	10:	//*****ClearUp****
		//Interpreter stoppen
		fbItpStartStopEx(bStart:= FALSE, bStop:= TRUE, sNciToPlc:= stGCodeRef.sNciToPlc);
		IF NOT fbItpStartStopEx.bBusy THEN
			IF fbItpStartStopEx.bErr THEN
				stError.ErrorId := UDINT_TO_UINT(fbItpStartStopEx.nErrId);
				nStateA_Common := 99;
			ELSE
				nStateA_Common := 11;
				fbFastMFunc.M_StopPrintAction(stGCodeRef.pCurrentTool,0);
				IF stGCodeRef.pCurrentTool > 0 THEN
					IF stGCodeRef.pCurrentTool^.P_eObjectType = E_ObjectType.OBJECTTYPE_VermesDisp THEN
						//Druck ausschalten
						MEMSET(ADR(stActionData),0,SIZEOF(stActionData));
						stActionData.eAction := E_Action.ACTION_SwitchPressure;
						stActionData.aParams[1] := 1;
						stGCodeRef.pCurrentTool^.M_ExeAction(stActionData);
					END_IF				
				END_IF
			END_IF
			IF pHighVoltTray > 0 THEN
				IF pHighVoltTray^.P_bPwrCutOffTriggered THEN
					nStateA_CommonNext := 30;	//In Parking-Pos fahren
				END_IF
				//Strom-Überwachung ausschalten
				pHighVoltTray^.M_CurrentMonitoring(FALSE);
			END_IF	
			fbItpStartStopEx(bStart:= FALSE, bStop:= FALSE, sNciToPlc:= stGCodeRef.sNciToPlc);
		END_IF
		
	11:	//Interpreter resetten (nötig, um Interpolationsgruppe zu löschen)
		fbItpResetEx2(bExecute:= TRUE, sNciToPlc:= stGCodeRef.sNciToPlc);
		IF NOT fbItpResetEx2.bBusy THEN
			IF fbItpResetEx2.bErr THEN
				stError.ErrorId := UDINT_TO_UINT(fbItpResetEx2.nErrId);
				nStateA_Common := 99;
			ELSE
				nStateA_Common := 20;
			END_IF
			fbItpResetEx2(bExecute:= FALSE, sNciToPlc:= stGCodeRef.sNciToPlc);
		END_IF
			
	20:	//Interpolationsgruppe löschen
		fbClearGroup(stGCodeRef:= stGCodeRef, bReGearInSlave:= TRUE, bExecute:= TRUE);
		IF NOT fbClearGroup.bBusy THEN
			IF fbClearGroup.bError THEN
				stError.ErrorId := fbClearGroup.nErrorId;
				nStateA_Common := 99;
			ELSE
				nStateA_Common := nStateA_CommonNext;
			END_IF
			fbClearGroup(stGCodeRef:= stGCodeRef, bExecute:= FALSE);
		END_IF
		
	30:	//In Parking-Pos fahren (MoveAllHome)
		MEMSET(ADR(stActionData),0,SIZEOF(stActionData));
		stActionData.eAction := E_Action.ACTION_MoveAllHome;
		stError.ErrorId := fbComplexAction.M_ExeAction(stActionData);
		IF stError.ErrorId > 0 THEN
			nStateA_Common := 99;
		ELSE
			nStateA_Common := 31;
		END_IF
		
	31: //MoveAllHome ready?
		IF NOT fbComplexAction.bBusy THEN
			IF fbComplexAction.bError THEN
				nStateA_Common := 99;
			ELSE
				nStateA_Common := 80;
			END_IF
		END_IF

END_CASE

IF nStateA_Common = 99 THEN
	stError.POUAction := E_POUACT.POUACT_A_Run;
	fbErrorList.M_Add(stError);
END_IF
END_ACTION

ACTION A_Start:
stError.POUState := nStateA_Common;

CASE nStateA_Common OF
	0:	//Interpolationsgruppe bilden
		stError.ErrorId := 0;
		fbBuildGroup(stGCodeRef:= stGCodeRef, bExecute:= TRUE);
		IF NOT fbBuildGroup.bBusy THEN
			IF fbBuildGroup.bError THEN
				stError.ErrorId := fbBuildGroup.nErrorId;
				nStateA_Common := 99;
			ELSE
				nStateA_Common := 1;
			END_IF
			fbBuildGroup(stGCodeRef:= stGCodeRef, bExecute:= FALSE);
		END_IF
		
		//Tools iterieren, in ToolAssigTable eintragen und gleich das MES-Tool ermitteln, welches im nächsten Schritt
		//eventuell vom Freifahren ausgeschlossen wird
	1:  pGCodeTool := 0;
		pMesCartDisp := 0;
		pHighVoltTray := pTarget^.M_GetFirstParentOfType(E_ObjectType.OBJECTTYPE_HighVoltTray);
		memset(ADR(GCode.stGCodeRef.aToolTable),0, SIZEOF(ST_GCodeTool) * GCode.cMaxGCodeTools);
		stGCodeRef.pHead^.P_pObjCollectNode^.nodes.M_GetIterator(iterDeep);
		WHILE iterDeep.pNode > 0 DO
			IF iterDeep.pNode^.P_pObject > 0 AND_THEN iterDeep.pNode^.P_pObject^.M_bIsGroup(E_ObjectGroup.OBJECTGROUP_MzTool) THEN
				pTempTool := iterDeep.pNode^.P_pObject;
				IF fbObjectDirectory.M_ObjIsGCodeTool(pTempTool^.P_nObjectID) THEN //GCodeTool?
					pGCodeTool := pTempTool;
					IF pGCodeTool^.P_nGCodeToolNr > 0 THEN
						IF pGCodeTool^.P_nGCodeToolNr <= cMaxGCodeTools THEN
							IF stGCodeRef.aToolTable[pGCodeTool^.P_nGCodeToolNr].pMzTool = 0 THEN
								stGCodeRef.aToolTable[pGCodeTool^.P_nGCodeToolNr].pMzTool := pGCodeTool;
								//MES-Kartusche und MES-Tray vorhanden?
								IF (pGCodeTool^.P_eObjectType = E_ObjectType.OBJECTTYPE_CartDispenser OR
									pGCodeTool^.P_eObjectType = E_ObjectType.OBJECTTYPE_CartDispStirrer) AND pHighVoltTray > 0 THEN
									pMesCartDisp := pGCodeTool;
									IF NOT pMesCartDisp^.P_bIsMESTool THEN
										//befindet sich MES-Kartusche über MES-Tray? Diese würde vom Freifahren ausgeschlossen
										IF NOT F_PointInnerRect(pMesCartDisp^.P_stCurrentPosPhys,pHighVoltTray^.P_stAbsRect) THEN
											pMesCartDisp := 0;	
										END_IF
									END_IF
								END_IF
								//Checken, ob Tool bereit für den Start im GCode-Mode
								stError.ErrorId := pGCodeTool^.M_CheckGCodeStart();
								IF stError.ErrorId > 0 THEN
									stError.ObjectId := pGCodeTool^.P_nObjectID;
									EXIT;
								END_IF
							ELSE
								//schon belegt, zwei Tools haben die gleiche ToolNr
								//sollte eigentlich schon in der GUI abgefangen werden
								stError.ErrorId := E_ErrorIdGCode.ERRORID_InvalidToolNr;
								EXIT;			
							END_IF
						ELSE
							//ToolNr zu groß
							//sollte eigentlich schon in der GUI abgefangen werden
							stError.ErrorId := E_ErrorIdGCode.ERRORID_InvalidToolNr;
							EXIT;			
						END_IF
					END_IF					
				END_IF
			END_IF
			iterDeep.M_Increment();
		END_WHILE
		
		//GCodeTargetNummern in TargetTable eintragen
		memset(ADR(GCode.stGCodeRef.aTargetTable),0, SIZEOF(UINT) * GCode.cMaxGCodeTargets);
		//wie komme ich hier an die Workplate ran?
		//über den Head und die zugeordnete Workplate
		stGCodeRef.pHead^.P_pAssignWorkplate^.P_pObjCollectNode^.nodes.M_GetIterator(iterDeep);
		WHILE iterDeep.pNode > 0 DO
			(* 1. Finde ein Objekt im Tree 2. Muss ein mögliches Target sein 3. Diese Objekt muss die gleiche Obj Id haben wie der in der GUI ausgewählte Print Point *)
			IF iterDeep.pNode^.P_pObject > 0  AND_THEN iterDeep.pNode^.P_pObject^.M_bIsGroup(E_ObjectGroup.OBJECTGROUP_Target) AND iterDeep.pNode^.P_pObject^.P_nObjectID = stInfo2.nTargetObjId THEN
				pTarget := iterDeep.pNode^.P_pObject;
				IF pTarget^.P_nGCodeTargetNr > 0 THEN
					//darf nicht größe als 20 sein 
					IF  pTarget^.P_nGCodeTargetNr > GCode.cMaxGCodeTargets THEN
						{warnig 'Imlement proper ErrorID'}
						stError.ErrorId := E_ErrorIdGCode.ERRORID_InvalidToolNr;
						RETURN;
					END_IF
					//darf noch nicht belegt sein
					IF GCode.stGCodeRef.aTargetTable[pTarget^.P_nGCodeTargetNr] > 0 THEN
						{warnig 'Imlement proper ErrorID'}
						stError.ErrorId := E_ErrorIdGCode.ERRORID_InvalidToolNr;
						RETURN;
					END_IF
					GCode.stGCodeRef.aTargetTable[pTarget^.P_nGCodeTargetNr] := pTarget^.P_nObjectID;
				END_IF
			END_IF
			iterDeep.M_Increment();
		END_WHILE
	
		//Tools freifahren
		IF stError.ErrorId = 0 THEN
			stError.ErrorId := stGCodeRef.pHead^.M_MoveFree(pMesCartDisp);
			IF stError.ErrorId > 0 THEN
				stError.ObjectId := stGCodeRef.pHead^.P_nObjectID;
				nStateA_Common := 99;
			ELSE
				nStateA_Common := 2;
			END_IF
		ELSE
			nStateA_Common := 99;
		END_IF
	
	2:	//Tools frei?
		IF NOT stGCodeRef.pHead^.M_GetActionBusy(E_Action.ACTION_MoveZ) THEN
			nStateA_Common := 3;
		END_IF
		
		IF stGCodeRef.pHead^.P_bError THEN
			stError.ErrorId := stGCodeRef.pHead^.P_nErrorId;
			stError.ObjectId := stGCodeRef.pHead^.P_nObjectID;
			nStateA_Common := 99;
		END_IF
	
	3:	//XY-Nullpunktverschiebung schreiben
		fbItpWriteZeroShiftEx(bExecute:= TRUE, sNciToPlc:= stGCodeRef.sNciToPlc, nZsNo:= 54, sZeroShiftDesc:= stGCodeRef.sZeroShiftDesc);	
		IF NOT fbItpWriteZeroShiftEx.bBusy THEN
			IF fbItpWriteZeroShiftEx.bErr THEN
				stError.ErrorId := UDINT_TO_UINT(fbItpWriteZeroShiftEx.nErrId);
				nStateA_Common := 99;
			ELSE
				stGCodeRef.pCurrentTool := 0;
				fbFastMFunc.M_Reset();
				fbHskMFunc.M_Reset();
				nStateA_Common := 4;
			END_IF
			fbItpWriteZeroShiftEx(bExecute:= FALSE, sNciToPlc:= GCode.stGCodeRef.sNciToPlc, nZsNo:= 54, sZeroShiftDesc:= stGCodeRef.sZeroShiftDesc);
		END_IF
		
	4: //RParameter 101 bis 125 löschen
		fbItpWriteRParams(bExecute:= TRUE, pAddr:= ADR(aRParamInit), nIndex:= 101 , nCount:= 25, sNciToPlc:= stGCodeRef.sNciToPlc); 
		IF NOT fbItpWriteRParams.bBusy THEN
			fbItpWriteRParams(bExecute:= FALSE, sNciToPlc:= stGCodeRef.sNciToPlc);
			lrAngle := pTarget^.P_lrAbsAngle;
			stGCodeRef.fbLimitCuboid.P_lrAngle := lrAngle;
			nStateA_Common := 5;
		END_IF
		
	5: //Verdrehwinkel des Targets in R126 schreiben (Winkel wird einen Schritt vorher ermittelt
		fbItpWriteRParams(bExecute:= TRUE, pAddr:= ADR(lrAngle), nIndex:= 126 , nCount:= 1, sNciToPlc:= stGCodeRef.sNciToPlc);
		IF NOT fbItpWriteRParams.bBusy THEN
			fbItpWriteRParams(bExecute:= FALSE, sNciToPlc:= stGCodeRef.sNciToPlc);
			nStateA_Common := 6;
		END_IF

	6:	//Interpreter starten
		fbItpStartStopEx(bStart:= TRUE,	bStop:= FALSE, sNciToPlc:= GCode.stGCodeRef.sNciToPlc);
		IF NOT fbItpStartStopEx.bBusy THEN
			IF fbItpStartStopEx.bErr THEN
				stError.ErrorId := UDINT_TO_UINT(fbItpStartStopEx.nErrId);
				nStateA_Common := 99;
			ELSE
				nStateA_Common := 7;
			END_IF
			fbItpStartStopEx(bStart:= FALSE, bStop:= FALSE, sNciToPlc:= GCode.stGCodeRef.sNciToPlc);
		END_IF
END_CASE

IF nStateA_Common = 7 THEN
	//Abfrage  des InterpreterStatus
	//Wechsel des States von Ready auf einen anderen State -> weiter zu A_Running
	//Nach dem Laden des Programms geht der Interpreter in Ready
	stInfo.nNciState := ItpGetStateInterpreter(GCode.stGCodeRef.sNciToPlc);
	IF stInfo.nNciState <> Tc2_NCI.NCI_INTERPRETER_READY THEN
		IF pHighVoltTray > 0 THEN
			//Strom-Überwachung einschalten
			pHighVoltTray^.M_CurrentMonitoring(TRUE);
		END_IF
		stGCodeRef.lrNcOverride := 100.0;
		nStateA_Common := 80;
	END_IF
END_IF

//Achtung, Implementation von Cancel ist hier schon wichtig!!!

IF nStateA_Common = 99 THEN
	stError.POUAction := E_POUACT.POUACT_A_Start;
	fbErrorList.M_Add(stError);
END_IF
END_ACTION

METHOD M_ClearGroup : ST_MethResult

VAR_INPUT
	bReGearIn : BOOL;
END_VAR
IF pXDrive = 0 OR pYDrive = 0 THEN	//GCode-Modul wurde noch nicht gestartet und folglich kann auch keine Gruppe vorhanden sein
	RETURN;
END_IF
M_ClearGroup.bBusy := TRUE;
fbClearGroup(stGCodeRef:= stGCodeRef, bReGearInSlave:= bReGearIn, bExecute:= TRUE);
IF NOT fbClearGroup.bBusy THEN
	IF fbClearGroup.bError THEN
		M_ClearGroup.bError := TRUE;
		M_ClearGroup.nErrorId := fbClearGroup.nErrorId;
	END_IF
	M_ClearGroup.bBusy := FALSE;
	fbClearGroup(stGCodeRef:= stGCodeRef, bExecute:= FALSE);
END_IF
END_METHOD

METHOD M_Continue : ERRORID
VAR_INPUT
END_VAR
IF nState = 6 THEN
	eGCodeState := E_GCodeState.GCodeState_ContinueRequest;
	nState := 7;
END_IF
END_METHOD

METHOD M_Pause : ERRORID
VAR_INPUT
END_VAR
IF stInfo.eGCodeState = E_GCodeState.GCodeState_Running AND nStateA_Common = 0 THEN
	IF pHighVoltTray > 0 THEN
		//Strom-Überwachung ausschalten
		pHighVoltTray^.M_CurrentMonitoring(FALSE);
	END_IF
	nState := 5;
END_IF
END_METHOD

METHOD M_Reset
VAR_INPUT
END_VAR
IF nState = 99 THEN
	nState := 60;
END_IF
END_METHOD

METHOD M_SetSequenceIds
VAR_INPUT
	pIdArray : POINTER TO ARRAY[1..5] OF DINT;
END_VAR
MEMCPY(ADR(stGCodeRef.aSequenceIds),pIdArray,20);
END_METHOD

METHOD M_SetStartZeroPoint : ERRORID
VAR_INPUT
	nTargetObjId 	: UINT;
	eTargetRef		: E_TargetRef;
	nCol			: UINT;
	nRow			: UINT;
	nZOffset		: DINT;
	nPausePointObjId: UINT;
	rHeight			: REAL;
END_VAR

VAR
	pMtp		: POINTER TO FB_Mtp;
	stPosTemp	: ST_3DPoint;
	rHeightTemp	: REAL;
END_VAR
CASE fbObjectDirectory.M_GetObjType(nTargetObjId) OF
	E_ObjectType.OBJECTTYPE_Point, E_ObjectType.OBJECTTYPE_Slide:
		//als TargetRef wird hier immer Mitte angenommen
		pTarget := fbObjectDirectory.M_GetObjPointer(nTargetObjId);
		stGCodeRef.stStartPos := pTarget^.M_GetAbsPos(0,E_TargetRef.TARGETREF_Center,0,0,0,1,nErrorId=> M_SetStartZeroPoint);
		GCode.stInfo2.nTargetObjId := nTargetObjId;
		
	E_ObjectType.OBJECTTYPE_Mtp:
		pTarget := fbObjectDirectory.M_GetObjPointer(nTargetObjId);
		IF eTargetRef <> E_TargetRef.TARGETREF_TwoDimArray THEN
			M_SetStartZeroPoint := E_ErrorIdCmd.ERRORID_InvalidTargetPointRef;
			RETURN;
		END_IF
		pMtp := pTarget;
		stGCodeRef.stStartPos := pMtp^.M_GetAbsPos(0,eTargetRef, nCol, nRow, 0, 1, nErrorId=> M_SetStartZeroPoint);
		IF M_SetStartZeroPoint > 0 THEN
			RETURN;
		END_IF
ELSE
	M_SetStartZeroPoint := E_ErrorIdCmd.ERRORID_UnsuitableTarget;
	RETURN;
END_CASE

stGCodeRef.fbLimitCuboid.P_stRefPoint := stGCodeRef.stStartPos;

stGCodeRef.pWaitPoint := 0;
IF nPausePointObjId > 0 THEN
	IF fbObjectDirectory.M_GetObjType(nPausePointObjId) = E_ObjectType.OBJECTTYPE_Point THEN
		stGCodeRef.pWaitPoint := fbObjectDirectory.M_GetObjPointer(nPausePointObjId);
	ELSE
		M_SetStartZeroPoint := E_ErrorIdGCode.ERRORID_InvalidPausePoint;
		RETURN;
	END_IF
END_IF

//Es kann nur der obere Head GCode ausführen
stGCodeRef.pHead := fbObjectDirectory.M_GetTopHead();

pXDrive := stGCodeRef.pHead^.P_pXDrive;
pYDrive := stGCodeRef.pHead^.P_pYDrive;

//Da hier noch kein Tool ausgewählt ist, bezieht sich Nullpunktverschiebung in XY bezieht sich vorerst den Head
//Bei der Toolauswahl wird entsprechend verrechnet 
stPosTemp := F_Sub3DPoints(stGCodeRef.stStartPos, stGCodeRef.pHead^.P_stAbsPosTotal);
stGCodeRef.sZeroShiftDesc.fShiftX := stPosTemp.X / 1000.0;
stGCodeRef.sZeroShiftDesc.fShiftY := stPosTemp.Y / 1000.0;
stGCodeRef.sZeroShiftDesc.fShiftZ := (stGCodeRef.stStartPos.Z + DINT_TO_REAL(nZOffset)) / 1000.0;
END_METHOD

METHOD M_ShiftZPos : ERRORID
VAR_INPUT
	rValue : REAL;
END_VAR
//Wird nur verschoben, wenn in Running oder Pause
IF (NOT bWriteZeroShift) AND (eGCodeState = E_GCodeState.GCodeState_Running OR eGCodeState = E_GCodeState.GCodeState_Pause) THEN
	stGCodeRef.sZeroShiftDesc.fShiftZ := stGCodeRef.sZeroShiftDesc.fShiftZ + (rValue / 1000.0);
	bWriteZeroShift := TRUE;
END_IF
END_METHOD

METHOD M_Start : ERRORID
VAR_INPUT
	sFileNumber : STRING;
END_VAR
//Kann nur aus dem State "Idle" ausgeführt werden
IF stInfo.eGCodeState = E_GCodeState.GCodeState_Idle THEN
	{IF defined(WIN10)}
	sGCodeFile := CONCAT(cPathWIN_10, sFileNumber);
	{ELSE}
	sGCodeFile := CONCAT(cPathWIN_EMBEDDED, sFileNumber);
	{END_IF}
	sGCodeFile := CONCAT(sGCodeFile,'.nc');
	bStop := FALSE;
	nState := 2;
	stInfo.eGCodeState := eGCodeState := E_GCodeState.GCodeState_Loading;
	stInfo.nFileNr := STRING_TO_UDINT(sFileNumber);
ELSE
	M_Start := E_ErrorIdGCode.ERRORID_InvalidNciState;
END_IF
END_METHOD

METHOD M_Stop
VAR_INPUT
END_VAR
IF nState > 1 THEN //Idle
	bStop := TRUE;
END_IF
END_METHOD

PROPERTY P_bMoveActionsLocked : BOOL
GET
P_bMoveActionsLocked := bMoveActionsLocked;
END_GET
SET
bMoveActionsLocked := P_bMoveActionsLocked;
END_SET
END_PROPERTY

PROPERTY P_bNciAvailable : BOOL
GET
P_bNciAvailable := bNciAvailable;
END_GET
END_PROPERTY

PROPERTY P_nProgress : UINT
GET
P_nProgress := nProgress;
END_GET
END_PROPERTY

END_PROGRAM

// ---- Hardware/XYDrive/FB_XYDriveBase.TcPOU
FUNCTION_BLOCK FB_XYDriveBase EXTENDS FB_HwModule
VAR PERSISTENT
	rRefPosMaster		: REAL;
	rWorkplateLength 	: REAL;
	rNullPosDist 		: REAL;
	rMaxPosDist 		: REAL;
	rSetupPosDist 		: REAL;
	rLimitMargeNeg 		: REAL;
	rLimitMargePos 		: REAL;
	rMaxSpeed 			: REAL;
	bSetupOK 			: BOOL; //Setup wurde durchgeführt	
	bInvertInitDir 		: BOOL; //Richtung bei Initialisierung umkehren(negativ)
END_VAR

VAR
	nErrorId 			: ERRORID;
	rActPos				: REAL;
	bHomed				: BOOL;
	
	eXYOrientation		: E_XYOrientation;

	bWriteAxisParameter : BOOL;
	nStateA_WriteAxisParamter : USINT;
	nStateWriteLimitNegative : USINT;
	nStateWriteLimitPositive : USINT;
	nStateWriteNCIFastSpeed : USINT;

	bSetup : BOOL;
	nStateA_Setup : USINT;
	bSetupWaitForResp : BOOL;
	bContinueSetup : BOOL;
	bSetupError: BOOL;
	
	bInit : BOOL;
	nStateA_Init : USINT;
	bReInit : BOOL;
	rHomePos : REAL;
	Delay : TON;
	bStopInit : BOOL;
	
	bJog : BOOL;
	nStateA_Jog : USINT;
	bJogForward : BOOL;
	bJogBackward : BOOL;
	bJogInching : BOOL;
	tmrJog : TON;	
	
	bMoveAbs : BOOL;
	nStateMoveAbs : USINT;
	bMoveRel : BOOL;
	nStateMoveRel : USINT;
	
	bCapture : BOOL;
	nStateA_Capture : USINT;
	bStopCapture : BOOL;
	nStateA_StopCapture : USINT;
	bCaptureOk 			: BOOL;
	bCaptureStopped 	: BOOL;
	rCapturedPos		: REAL;
	
	bStop	: BOOL;
	nStateA_Stop : USINT;
	
	bReset : BOOL;
	nStateA_Reset : USINT;
	
	nStateA_Error : USINT;
	
	pMultiZRef : POINTER TO FB_MultiZRef;
	
	stAdsAddress : ST_AdsAdress;
	
	rTrigError	: R_TRIG;

END_VAR


IF bWriteAxisParameter THEN
	A_WriteAxisParameter();
	IF nStateA_WriteAxisParamter >= 80 THEN
		IF nStateA_WriteAxisParamter >= 99 THEN
			bError := TRUE;
		END_IF
		nStateA_WriteAxisParamter := 0;
		bWriteAxisParameter := FALSE;
	END_IF
END_IF

IF bSetup THEN
	A_Setup();
	IF nStateA_Setup >= 80 THEN
		IF nStateA_Setup >= 99 THEN
			bError := TRUE;
		END_IF
		nStateA_Setup := 0;
		bSetup := FALSE;
	END_IF
END_IF

IF bInit THEN
	A_Init();
	IF nStateA_Init = 80 THEN
		nStateA_Init := 0;
		bInit := FALSE;
	END_IF

	IF nStateA_Init = 99 THEN	//Error
		nStateA_Init := 0;
		bInit := FALSE;
		bError := TRUE;
	END_IF
END_IF

IF bMoveAbs THEN
	A_MoveAbs();
	IF nStateMoveAbs >= 80 THEN
		IF nStateMoveAbs >= 99 THEN	//Error
			bError := TRUE;
		END_IF
		nStateMoveAbs := 0;
		bMoveAbs := FALSE;
	END_IF	
END_IF

IF bMoveRel THEN
	A_MoveRel();
	IF nStateMoveRel >= 80 THEN
		IF nStateMoveRel >= 99 THEN	//Error
			bError := TRUE;
		END_IF
		nStateMoveRel := 0;
		bMoveRel := FALSE;
	END_IF	
END_IF

IF bJog THEN
	A_Jog();
	IF nStateA_Jog >= 80 THEN
		IF nStateA_Jog >= 99 THEN	//Error
			bError := TRUE;
		END_IF
		nStateA_Jog := 0;
		bJog := FALSE;
	END_IF	
END_IF

IF bCapture THEN
	A_Capture();
	IF nStateA_Capture >= 80 THEN
		IF nStateA_Capture >= 99 THEN	//Error
			bError := TRUE;
		END_IF
		nStateA_Capture := 0;
		bCapture := FALSE;
	END_IF	
END_IF

IF bStopCapture THEN
	A_StopCapture();
	IF nStateA_StopCapture >= 80 THEN
		IF nStateA_StopCapture >= 99 THEN	//Error
			bError := TRUE;
		END_IF
		nStateA_StopCapture := 0;
		bStopCapture := FALSE;
	END_IF	
END_IF

IF bReset THEN
	A_Reset();
	IF nStateA_Reset >= 80 THEN
		IF nStateA_Reset >= 99 THEN
			bError := TRUE;
		END_IF
		nStateA_Reset := 0;
		bReset := FALSE;
	END_IF
END_IF

IF bError THEN
	A_Error();
END_IF

IF NOT (bInit OR bMoveAbs OR bMoveRel OR bJog OR bReset OR bSetup) THEN
	bStop := FALSE;
	bBusy := FALSE;
ELSE
	bBusy := TRUE;
END_IF

rTrigError(CLK:= bError);
IF rTrigError.Q THEN
	stError.ErrorId := nErrorId;
	fbErrorList.M_Add(stError);
END_IF

PROPERTY P_bHomed : BOOL
GET
P_bHomed := bHomed;
END_GET
END_PROPERTY

ACTION A_Setup:

END_ACTION

METHOD M_GetProperty : ERRORID
VAR_INPUT
	eType	: E_HardwarePropType;
END_VAR
VAR_OUTPUT
	nValue 	: DINT;
END_VAR
CASE eType OF
	E_HardwarePropType.RefPos1:
		nValue := REAL_TO_DINT(rRefPosMaster);
	E_HardwarePropType.MinPos:
		nValue := REAL_TO_DINT(P_rMinPos);
	E_HardwarePropType.MaxPos:
		nValue := REAL_TO_DINT(P_rMaxPos);
	E_HardwarePropType.LimitMargeNeg:
		nValue := REAL_TO_DINT(rLimitMargeNeg);
	E_HardwarePropType.LimitMargePos:
		nValue := REAL_TO_DINT(rLimitMargePos);
	E_HardwarePropType.MaxSpeed:
		nValue := REAL_TO_DINT(rMaxSpeed);
	E_HardwarePropType.WorkplateDim:
		nValue := REAL_TO_DINT(rWorkplateLength);
	E_HardwarePropType.NullPosDist:
		nValue := REAL_TO_DINT(rNullPosDist);
	E_HardwarePropType.MaxPosDist:
		nValue := REAL_TO_DINT(rMaxPosDist);
	E_HardwarePropType.SetupPosDist:
		nValue := REAL_TO_DINT(rSetupPosDist);
	E_HardwarePropType.InvertInitDir:
		nValue := BOOL_TO_DINT(bInvertInitDir);		
ELSE
	M_GetProperty := E_ErrorIdCmd.ERRORID_InvalidHwProperty;	
END_CASE
END_METHOD

METHOD M_Init : ERRORID
VAR_INPUT
	bReInit : BOOL;
END_VAR
IF bBusy THEN
	M_Init := E_ErrorIdCmd.ERRORID_AxisStillBusy;
ELSE
	THIS^.bReInit := bReInit;
	//Die Action wird von hier aus einmalig ausgeführt damit ein Aufruf schon in diesem Zyklus stattfindet
	rHomePos := rRefPosMaster;
	bInit := TRUE;
	A_Init();		
END_IF
END_METHOD

METHOD M_PowerOn : ERRORID
VAR_INPUT
END_VAR
END_METHOD

METHOD M_MoveRel : ERRORID
VAR_INPUT
	rDistance		: REAL;
	rSpeed			: REAL;
	rAcceleration 	: REAL;
	rDeceleration 	: REAL;	
END_VAR
END_METHOD

ACTION A_Reset:

END_ACTION

PROPERTY P_bIsTwinDrive : BOOL
GET
END_GET
END_PROPERTY

METHOD M_Stop : ERRORID
VAR_INPUT
END_VAR
IF bBusy AND NOT bStop THEN
	bStop := TRUE;
END_IF
END_METHOD

METHOD M_Setup : ERRORID
VAR_INPUT
END_VAR
IF bBusy THEN
	M_Setup := E_ErrorIdCmd.ERRORID_AxisStillBusy;
ELSE
	THIS^.bReInit := TRUE;
	rHomePos := 0;
	bSetup := TRUE;
END_IF
END_METHOD

PROPERTY P_nErrorId : ERRORID
GET
P_nErrorId := nErrorId;
END_GET
END_PROPERTY

METHOD M_PowerOff : ERRORID
VAR_INPUT
END_VAR
END_METHOD

PROPERTY P_bIsMoving : BOOL
GET
END_GET
END_PROPERTY

ACTION A_Error:

END_ACTION

PROPERTY P_pAxisRef : POINTER TO AXIS_REF
GET
END_GET
END_PROPERTY

ACTION A_Init:

END_ACTION

METHOD M_StopCapture : ERRORID
VAR_INPUT
END_VAR
bStopCapture := TRUE;
bCaptureStopped := FALSE;
A_StopCapture();
END_METHOD

METHOD M_SetProperty : ERRORID
VAR_INPUT
	eType	: E_HardwarePropType;
	nValue 	: DINT;
END_VAR
CASE eType OF
	E_HardwarePropType.RefPos1:
		rRefPosMaster := DINT_TO_REAL(nValue);
	E_HardwarePropType.MinPos:
		M_SetProperty := E_ErrorIdCmd.ERRORID_OnlyReadHwProp;
	E_HardwarePropType.MaxPos:
		M_SetProperty := E_ErrorIdCmd.ERRORID_OnlyReadHwProp;
	E_HardwarePropType.LimitMargeNeg:
		rLimitMargeNeg := DINT_TO_REAL(nValue);
		bWriteAxisParameter := TRUE;
	E_HardwarePropType.LimitMargePos:
		rLimitMargePos := DINT_TO_REAL(nValue);
		bWriteAxisParameter := TRUE;
	E_HardwarePropType.MaxSpeed:
		rMaxSpeed := DINT_TO_REAL(nValue);
		bWriteAxisParameter := TRUE;
	E_HardwarePropType.WorkplateDim:
		rWorkplateLength := DINT_TO_REAL(nValue);
		bWriteAxisParameter := TRUE;
	E_HardwarePropType.NullPosDist:
		rNullPosDist := DINT_TO_REAL(nValue);
		bWriteAxisParameter := TRUE;
	E_HardwarePropType.MaxPosDist:
		rMaxPosDist := DINT_TO_REAL(nValue);
		bWriteAxisParameter := TRUE;
	E_HardwarePropType.SetupPosDist:
		rSetupPosDist := DINT_TO_REAL(nValue);
	E_HardwarePropType.InvertInitDir:
		bInvertInitDir := DINT_TO_BOOL(nValue);
ELSE
	M_SetProperty := E_ErrorIdCmd.ERRORID_InvalidHwProperty;	
END_CASE
END_METHOD

METHOD M_GearOut : ST_MethResult
END_METHOD

PROPERTY P_tHomingTime : TIME
GET
//nur aus Kompatibilitätsgründen PlattformD impl.
P_tHomingTime := T#0s;
END_GET
END_PROPERTY

METHOD M_Capture : ERRORID
VAR_INPUT
END_VAR
END_METHOD

PROPERTY P_stAdsAddress : ST_AdsAdress
SET
stAdsAddress := P_stAdsAddress;
END_SET
GET
P_stAdsAddress := stAdsAddress;
END_GET
END_PROPERTY

PROPERTY P_bHasJob : BOOL
GET
END_GET
END_PROPERTY

PROPERTY P_bCoupled : BOOL
GET
END_GET
END_PROPERTY

ACTION A_Capture:

END_ACTION

PROPERTY P_bHoming : BOOL
GET
P_bHoming := bInit;
END_GET
END_PROPERTY

PROPERTY P_bSetupWaitForResp : BOOL
GET
P_bSetupWaitForResp := bSetupWaitForResp;
END_GET
END_PROPERTY

METHOD FB_init : BOOL
VAR_INPUT
	bInitRetains 	: BOOL; // if TRUE, the retain variables are initialized (warm start / cold start)
	bInCopyCode 	: BOOL;  // if TRUE, the instance afterwards gets moved into the copy code (online change)
	eXYOrientation	: E_XYOrientation;
END_VAR
THIS^.eXYOrientation := eXYOrientation;
END_METHOD

METHOD M_Reset
VAR_INPUT
END_VAR
IF bError AND NOT bReset THEN
	bReset := TRUE;
END_IF
END_METHOD

ACTION A_StopCapture:

END_ACTION

METHOD M_ContinueSetup
VAR_INPUT
END_VAR
bContinueSetup := TRUE;
END_METHOD

ACTION A_WriteAxisParameter:

END_ACTION

PROPERTY P_rActPos : REAL
GET
P_rActPos := rActPos;
END_GET
END_PROPERTY

PROPERTY P_rMaxPos : REAL
GET
P_rMaxPos := rWorkplateLength - rNullPosDist - rMaxPosDist - rLimitMargePos;
END_GET
END_PROPERTY

METHOD M_Jog : ERRORID
VAR_INPUT
	bForward	: BOOL;
	bBackward	: BOOL;
	bInching	: BOOL;
	rDistance	: REAL;
	rSpeed		: REAL;		
END_VAR
END_METHOD

ACTION A_Jog:

END_ACTION

ACTION A_MoveRel:

END_ACTION

PROPERTY P_rMinPos : REAL
GET
P_rMinPos := rLimitMargeNeg;
END_GET
END_PROPERTY

METHOD M_MoveAbs : ERRORID
VAR_INPUT
	rPosition 		: REAL;
	rSpeed			: REAL;
	rAcceleration 	: REAL;
	rDeceleration 	: REAL;
END_VAR
END_METHOD

PROPERTY P_bCaptureOk : BOOL
GET
P_bCaptureOk := bCaptureOk;
END_GET
END_PROPERTY

METHOD M_GearIn : ST_MethResult
END_METHOD

PROPERTY P_pMultiZRef : POINTER TO FB_MultiZRef
SET
pMultiZRef := P_pMultiZRef;
END_SET
GET
P_pMultiZRef := pMultiZRef;
END_GET
END_PROPERTY

PROPERTY P_rMaxSpeed : REAL
GET
P_rMaxSpeed := rMaxSpeed;
END_GET
END_PROPERTY

METHOD M_SetProperties : ERRORID
VAR_INPUT
	refCmdData : REFERENCE TO ST_CmdData;
END_VAR
rWorkplateLength := DINT_TO_REAL(refCmdData.n32Data[1]);
rNullPosDist := DINT_TO_REAL(refCmdData.n32Data[2]);
rMaxPosDist := DINT_TO_REAL(refCmdData.n32Data[3]);
rSetupPosDist := DINT_TO_REAL(refCmdData.n32Data[4]);
bInvertInitDir := DINT_TO_BOOL(refCmdData.n32Data[5]);
END_METHOD

ACTION A_MoveAbs:

END_ACTION

PROPERTY P_rCapturedPos : REAL
GET
P_rCapturedPos := rCapturedPos;
END_GET
END_PROPERTY

PROPERTY P_bCaptureStopped : BOOL
GET
P_bCaptureStopped := bCaptureStopped;
END_GET
END_PROPERTY

PROPERTY P_bIsCoupled : BOOL
GET
END_GET
END_PROPERTY

PROPERTY P_eXYOrientation : E_XYOrientation
GET
P_eXYOrientation := eXYOrientation;
END_GET
SET
eXYOrientation := P_eXYOrientation;
END_SET
END_PROPERTY

END_FUNCTION_BLOCK

// ---- Hardware/MultiZ/FB_MultiZRef.TcPOU
FUNCTION_BLOCK FB_MultiZRef EXTENDS FB_CanNodeBase

VAR_INPUT
	aFbZAxisRef 	: ARRAY[1..7] OF FB_ZAxisRef(THIS);
	aFbPiezoRef		: ARRAY[1..7] OF FB_PiezoRef(THIS);
	aFbHeaterRef	: ARRAY[1..7] OF FB_MZHeaterRef(THIS);
	aFbExtruderRef	: ARRAY[1..7] OF FB_PistonExtruderRef(THIS);
	aFbGripperRef	: ARRAY[1..7] OF FB_GripperRef(THIS);
	stStampSupport 	: ST_StampSupport;
	stStrobTrigger	: ST_StrobTrigger; //Sdo
	aDigiOut		AT %Q* : ARRAY[1..7] OF BOOL;
	aFbGPInputRef	: ARRAY[1..6] OF FB_GPInputRef(THIS);
	bFixConfig		: BOOL;
	nErrorGlobal	AT %I* : USINT;
END_VAR

VAR
	i				: USINT;
	bLegacy			: BOOL;
	nAxisNr			: USINT;
	nAxisNrZSensor 	: USINT;
	
	//bPrepareAxis 			: BOOL;
	nStateA_PrepareAxis 	: USINT;
	nStateA_PrepareAxisNext : USINT;
	nPrepareAxisNr 			: USINT;
	nTemp					: UDINT;
	sTemp					: STRING;
	sHwIdTemp				: ST_HardwareId;
	nTriggerVersion			: USINT;
	nState					: USINT;
	
	//ResetError
	bMzBaseRestarted : BOOL;
	bGlobErrorReseted : BOOL;

	//A_SetConfig	
	bSetConfig : BOOL;
	nStateA_SetConfig : USINT;
	nStateA_SetConfigNext : USINT;
	bSetConfigEnable : BOOL;
	nStateA_ResetError : USINT;
	tmrTimeout : TON;
	nRemoteCRC : UINT;
	nLocalCRC : UINT;
	
	//A_Monitor()
	nStateA_Monitor 	: USINT;
	bGlobError 			: BOOL;
	fbSdoRead_Monitor 	: FB_SDO_READ;
	
END_VAR

VAR PERSISTENT
	stZSensorCalibration : ARRAY[1..4] OF ST_ZSensorCalibration;
END_VAR

IF bNodeEnabled THEN
	IF nState = 0 THEN //Preparing Step1 (Base)
		SUPER^();
		IF bPreparingOK THEN
			nPrepareAxisNr := 1;
			FOR i:= 1 TO 7 BY 1 DO
				IF NOT aFbZAxisRef[i].stInput.nStatus.3 THEN
					aFbZAxisRef[i].stOutput.nCtrl := 0;
					aFbZAxisRef[i].stOutput.nMode := 0;
					aFbZAxisRef[i].stOutput.nTrgtPos := 0;
					aFbZAxisRef[i].stOutput.nVelo := 0;
				END_IF
			END_FOR
			nState := 1;
		ELSIF bError THEN
			nState := 99;
		END_IF
	ELSIF nState = 1 THEN
		A_PrepareAxis();
		IF nStateA_PrepareAxis >= 80 THEN
			IF nStateA_PrepareAxis >= 99 THEN
				nState := 99;
				bError := TRUE;
			ELSE
				nState := 2;
			END_IF
			nStateA_PrepareAxis := 0;
		END_IF
	ELSIF nState = 2 THEN //Operational
		SUPER^(); //wird nur zur für ResetApp benötigt
		
		IF bSetConfig THEN
			IF bLegacy THEN
				A_SetConfigLegacy();	//alte Firmware ohne Toolerkennung
			ELSE
				A_SetConfig();
			END_IF
			IF nStateA_SetConfig >= 80 THEN
				IF nStateA_SetConfig >= 99 THEN
					bError := TRUE;
				END_IF
				nStateA_SetConfig := 0;
				bSetConfig := FALSE;
			END_IF
		END_IF
		
		IF bResetError THEN
			A_ResetError();
			IF nStateA_ResetError >= 80 THEN
				bError := FALSE;
				IF nStateA_ResetError >= 99 THEN
					bError := TRUE;
				END_IF
				nStateA_ResetError := 0;
				bResetError := FALSE;
			END_IF
		END_IF
		
	END_IF
	
	bBusy := (nState < 2) OR bSetConfig OR bResetError OR bResetApp;

	IF NOT (bBusy OR bStopMonitor) THEN
		A_Monitor();
	END_IF
	
END_IF

ACTION A_Monitor:
//Monitor CanNode
SUPER^.A_Monitor();

//Monitor GlobError
IF nStateA_Monitor = 0 THEN
	IF nErrorGlobal > 0 AND NOT bGlobError THEN
		bGlobError := TRUE;
		bError := TRUE;
		stError.HardwareGrp := E_HardwareGrp.MultiZBasis;
		stError.HardwareNr := stHardwareId.nItem;
		stError.POU := E_POU.POU_FB_MultiZRef;
		stError.POUAction := E_POUACT.POUACT_A_Monitor;
		stError.ErrorId := F_MultiZError_TO_ErrorId(nErrorGlobal);
		nStateA_Monitor := 2; //LastErrorState auslesen
	ELSE
		nStateA_Monitor := 1;
	END_IF
END_IF

//Monitor AxisError
IF nStateA_Monitor = 1 THEN
	nStateA_Monitor := 0;
	FOR nAxisNr := 1 TO 7 BY 1 DO
		IF aFbZAxisRef[nAxisNr].stInput.nStatus.7 THEN //Achse vorhanden?
			//Achse ist schon in Error -> dieser braucht nicht mehr gemeldet werden
			//Dieser Errorstatus kann auch durch Funktionsbausteine gesetzt werden, die auf eine
			//Achsenreferenz zugreifen. (z.B. FB_Zm_Home, FB_Zm_Jog usw.
			IF NOT aFbZAxisRef[nAxisNr].stStatus.bError THEN
				IF NOT aFbZAxisRef[nAxisNr].bIngoreError AND 
					(aFbZAxisRef[nAxisNr].stInput.nStatus.3 OR aFbZAxisRef[nAxisNr].stInput.nError > 0) THEN
					aFbZAxisRef[nAxisNr].stStatus.bError := TRUE;
					//Fehler melden	(nur 1x)
					stError.HardwareGrp := E_HardwareGrp.AxisZ;
					stError.HardwareNr := nAxisNr;
					stError.POU := E_POU.POU_FB_MultiZRef;
					stError.POUAction := E_POUACT.POUACT_A_Monitor;
					stError.ErrorId := F_MultiZError_TO_ErrorId(aFbZAxisRef[nAxisNr].stInput.nError);
					nStateA_Monitor := 2; //LastErrorState auslesen
					EXIT;
				END_IF
			END_IF
			IF aFbZAxisRef[nAxisNr].stStatus.bError THEN
				bError := TRUE;
			END_IF
		END_IF		
	END_FOR
END_IF

//Read LastErrorState
IF nStateA_Monitor = 2 THEN
	fbSdoRead_Monitor(sADSNetID:= stAdsAdress.sNetId, nPortNr:= stAdsAdress.nPort, 
				nIndex:= cLastErrorState.nIndex, nSubIndex:= cLastErrorState.nSubIndex,
				nDataLength:= cLastErrorState.nLength, bExecute:= TRUE);
	IF NOT fbSdoRead_Monitor.bBusy THEN
		stError.ErrorId2 := DINT_TO_UDINT(fbSdoRead_Monitor.nData);
		fbSdoRead_Monitor(bExecute:= FALSE);
		nStateA_Monitor := 3;
	END_IF
END_IF

//Notify Error
IF nStateA_Monitor = 3 THEN
	fbErrorList.M_Add(stError);
	nStateA_Monitor := 0;
END_IF
END_ACTION

ACTION A_PrepareAxis:
//1.Versionsvergleich -> Legacy
IF nStateA_PrepareAxis = 0 THEN
	IF F_CompVersion(sSoftwVersion,'1.10.X') = -1 THEN //alte Firmware ohne Toolerkennung
		bLegacy := TRUE;
	END_IF
	nStateA_PrepareAxis := 1;
END_IF

//2.Versionen der Motorsteuerungen auslesen
IF nStateA_PrepareAxis = 1 THEN
	//TMC-Version der Motorsteuerungen auslesen
	fbSdoRead(sADSNetID:= stAdsAdress.sNetId, nPortNr:= stAdsAdress.nPort,
			nIndex:= cTMCVersion.nIndex, nSubIndex:= nPrepareAxisNr, nDataLength:= cTMCVersion.nLength, bExecute:= TRUE); 
	
	IF NOT fbSdoRead.bBusy THEN
		IF fbSdoRead.bError THEN
			nErrorId := fbSdoRead.nAdsErrorId;
			nErrorId2 := fbSdoRead.nSdoErrorId;
			nStateA_PrepareAxis := 99;	//Error
		ELSE
			aFbZAxisRef[nPrepareAxisNr].nTmcModulId := DINT_TO_UINT(SHR(fbSdoRead.nData,16));
			nTemp := DINT_TO_UDINT(fbSdoRead.nData) AND 16#0000FF00;
			nTemp := SHR(nTemp,8);
			sTemp := UDINT_TO_STRING(nTemp);
			sTemp := CONCAT(sTemp,'.');
			nTemp := DINT_TO_UDINT(fbSdoRead.nData) AND 16#000000FF;
			sTemp := CONCAT(sTemp,UDINT_TO_STRING(nTemp));
			aFbZAxisRef[nPrepareAxisNr].sTmcVersion := sTemp;
			IF bLegacy THEN
				nStateA_PrepareAxis := 80;
			ELSE
				nStateA_PrepareAxis := 2;
			END_IF
			
			//Nächste aktive Achse für das Auslesen der TMC-Version ermitteln
			FOR nPrepareAxisNr := nPrepareAxisNr + 1 TO 7 BY 1 DO
				IF aFbZAxisRef[nPrepareAxisNr].stInput.nStatus.7 THEN
					//HwId Item auf ZAxis Parent Item übertragen
					aFbZAxisRef[nPrepareAxisNr].M_RenewHwId();
					nStateA_PrepareAxis := 1;
					EXIT;
				END_IF
			END_FOR
		END_IF
		fbSdoRead(bExecute:= FALSE);
	END_IF
END_IF

IF nStateA_PrepareAxis = 2 THEN
	IF bLegacy THEN
		nStateA_PrepareAxis := 80;
	ELSE
		nPrepareAxisNr := 1;
		nStateA_PrepareAxis := 3;
	END_IF
END_IF

//ToolTypes auslesen (nur bei Toolerkennung möglich) dafür muss bei SetConfig nicht mehr separat ausgelesen werden
IF nStateA_PrepareAxis = 3 THEN
	fbSdoRead(sADSNetID:= stAdsAdress.sNetId, nPortNr:= stAdsAdress.nPort,
			nIndex:= cToolType.nIndex, nSubIndex:= nPrepareAxisNr, nDataLength:= cToolType.nLength, bExecute:= TRUE);
			
	IF NOT fbSdoRead.bBusy THEN
		IF fbSdoRead.bError THEN
			nErrorId := fbSdoRead.nAdsErrorId;
			nErrorId2 := fbSdoRead.nSdoErrorId;
			nStateA_PrepareAxis := 99;	//Error
		ELSE
			aFbZAxisRef[nPrepareAxisNr].eDetectedToolType := DINT_TO_USINT(fbSdoRead.nData);
			nStateA_PrepareAxis := 4;
			//Nächste aktive Achse ermitteln
			FOR nPrepareAxisNr := nPrepareAxisNr + 1 TO 7 BY 1 DO
				IF aFbZAxisRef[nPrepareAxisNr].stInput.nStatus.7 THEN
					nStateA_PrepareAxis := 3;
					EXIT;
				END_IF
			END_FOR
		END_IF
		fbSdoRead(bExecute:= FALSE);
	END_IF	
END_IF

IF nStateA_PrepareAxis = 4 THEN
	nPrepareAxisNr := 1;
	nStateA_PrepareAxis := 5;
END_IF

//HeaterExits auslesen (nur bei Toolerkennung möglich) dafür muss bei SetConfig nicht mehr separat ausgelesen werden
IF nStateA_PrepareAxis = 5 THEN
	fbSdoRead(sADSNetID:= stAdsAdress.sNetId, nPortNr:= stAdsAdress.nPort,
			nIndex:= cHeaterExist.nIndex, nSubIndex:= nPrepareAxisNr, nDataLength:= cHeaterExist.nLength, bExecute:= TRUE);
			
	IF NOT fbSdoRead.bBusy THEN
		IF fbSdoRead.bError THEN
			nErrorId := fbSdoRead.nAdsErrorId;
			nErrorId2 := fbSdoRead.nSdoErrorId;
			nStateA_PrepareAxis := 99;	//Error
		ELSE
			aFbHeaterRef[nPrepareAxisNr].P_bHeaterDetected := DINT_TO_BOOL(fbSdoRead.nData);
			nStateA_PrepareAxis := 6;
			//Nächste aktive Achse ermitteln
			FOR nPrepareAxisNr := nPrepareAxisNr + 1 TO 7 BY 1 DO
				IF aFbZAxisRef[nPrepareAxisNr].stInput.nStatus.7 THEN
					nStateA_PrepareAxis := 5;
					EXIT;
				END_IF
			END_FOR
		END_IF
		fbSdoRead(bExecute:= FALSE);
	END_IF	
END_IF

IF nStateA_PrepareAxis = 6 THEN
	nPrepareAxisNr := 1;
	nStateA_PrepareAxis := 7;
END_IF

IF nStateA_PrepareAxis = 7 THEN	//Versionen der Tools auslesen
	fbSdoRead(sADSNetID:= stAdsAdress.sNetId, nPortNr:= stAdsAdress.nPort,
			nIndex:= cToolVersion.nIndex, nSubIndex:= nPrepareAxisNr, nDataLength:= cToolVersion.nLength, bExecute:= TRUE);
			
	IF NOT fbSdoRead.bBusy THEN
		IF fbSdoRead.bError THEN
			nErrorId := fbSdoRead.nAdsErrorId;
			nErrorId2 := fbSdoRead.nSdoErrorId;
			nStateA_PrepareAxis := 99;	//Error
		ELSE
			aFbZAxisRef[nPrepareAxisNr].nToolVersion := DINT_TO_USINT(fbSdoRead.nData);
			nStateA_PrepareAxis := 8;

			//Nächste aktive Achse für das Auslesen der TMC-Version ermitteln
			FOR nPrepareAxisNr := nPrepareAxisNr + 1 TO 7 BY 1 DO
				IF aFbZAxisRef[nPrepareAxisNr].stInput.nStatus.7 THEN
					nStateA_PrepareAxis := 7;
					EXIT;
				END_IF
			END_FOR
		END_IF
		fbSdoRead(bExecute:= FALSE);
	END_IF	
END_IF

//TriggerVersion auslesen
IF nStateA_PrepareAxis = 8 THEN
	fbSdoRead(sADSNetID:= stAdsAdress.sNetId, nPortNr:= stAdsAdress.nPort,
				nIndex:= cTriggerVersion.nIndex, nSubIndex:= cTriggerVersion.nSubIndex, nDataLength:= cTriggerVersion.nLength, bExecute:= TRUE);
			
	IF NOT fbSdoRead.bBusy THEN
		IF fbSdoRead.bError THEN
			nErrorId := fbSdoRead.nAdsErrorId;
			nErrorId2 := fbSdoRead.nSdoErrorId;
			nStateA_PrepareAxis := 99;	//Error
		ELSE
			nTriggerVersion := DINT_TO_USINT(fbSdoRead.nData);
			nStateA_PrepareAxis := 9;
		END_IF
		fbSdoRead(bExecute:= FALSE);
	END_IF	
END_IF

//SubAxis setzen (für den Fall dass an Achse 3 ein StampSupport sich befindet)
IF nStateA_PrepareAxis = 9 THEN
	IF aFbZAxisRef[3].eDetectedToolType = E_MzToolType.TOOL_TYPE_Stamp THEN
		aFbZAxisRef[4].bIsSubAxis := TRUE;
		aFbZAxisRef[5].bIsSubAxis := TRUE;
	END_IF
	nStateA_PrepareAxis := 80;
END_IF

IF nStateA_PrepareAxis = 99 THEN
	fbErrorList.M_AddExt(nErrorId:= nErrorId, nErrorId2:= nErrorId2, 
	HardwareGrp:= E_HardwareGrp.AxisZ, 
	HardwareNr:= nAxisNr, 
	POU:= E_POU.POU_FB_MultiZRef, 
	POUAction:= E_POUACT.POUACT_A_Init,
	POUState:= nPOUState);
	nErrorId2 := 0;
END_IF
END_ACTION

ACTION A_ResetApp:
IF nStateA_ResetApp = 0 THEN	//MultiZ resetten
	fbSdoWrite(sADSNetID:= stAdsAdress.sNetId, nPortNr:= stAdsAdress.nPort,
				nIndex := cUpdateRequest.nIndex, nSubIndex := 8, nDataLength := 1, nData:= 1, bExecute:= TRUE);
	IF NOT fbSdoWrite.bBusy THEN
		IF fbSdoWrite.bError THEN
			nErrorId := fbSdoWrite.nAdsErrorId;
			nErrorId2 := fbSdoWrite.nSdoErrorId;
			nStateA_ResetApp := 99;  //Error
		ELSE
			FOR i:= 1 TO 7 BY 1 DO
				aFbZAxisRef[i].stOutput.nMode := 0;
			END_FOR
			nStateA_ResetApp := 80;
		END_IF
		fbSdoWrite(bExecute:= FALSE);
	END_IF
END_IF
END_ACTION

ACTION A_ResetError:
nPOUState := nStateA_ResetError;
CASE nStateA_ResetError OF
	//**************************Begin CheckGlobError**********************************
	0:	//Node erreichbar?
		tmrTimeout(IN:= FALSE);
		nErrorId := 0;
		nErrorId2 := 0;
		IF nNodeState > 0 THEN
			CASE nNodeState OF
				1:	nErrorId := E_ErrorIdCan.ERRORID_NodeDeactivated;
				2:	nErrorId := E_ErrorIdCan.ERRORID_NodeNotFound;
				4:	nErrorId := E_ErrorIdCan.ERRORID_SdoSyntaxErrorAtStartup;
				5:	nErrorId := E_ErrorIdCan.ERRORID_SdoDataMismatchAtStartup;
				12:	nErrorId := E_ErrorIdCan.ERRORID_NodePreOP;
			END_CASE
			nStateA_ResetError := 99;
		ELSE
			//Restart Base erforderlich?
			IF (nErrorGlobal = 14 OR nErrorGlobal = 18 OR  nErrorGlobal = 255) THEN
				nStateA_ResetError := 20;	//RestartMzBase	
			ELSIF nErrorGlobal > 0 THEN
				nStateA_ResetError := 1;	//ResetGlobError
			ELSE
				nStateA_ResetError := 10;	//CheckAndResetAxisError
			END_IF
		END_IF
	//***************************End CheckGlobError***********************************

	//**************************Begin ResetGlobError**********************************
	1:	//globalen Fehler zurücksetzen
		IF bGlobErrorReseted OR bMzBaseRestarted THEN
			nErrorId := E_ErrorIdCmd.ERRORID_ErrorResetFailed;
			nErrorId2 := 0;
			nStateA_ResetError := 99;
			RETURN;
		END_IF
		fbSdoWrite(sADSNetID:= stAdsAdress.sNetId, nPortNr:= stAdsAdress.nPort,
					nIndex:= cGlobError.nIndex, nSubIndex:= cGlobError.nSubIndex, 
					nDataLength:= cGlobError.nLength, nData:= 0, bExecute:= TRUE);
		IF NOT fbSdoWrite.bBusy THEN
			IF fbSdoWrite.bError THEN
				nErrorId := fbSdoWrite.nAdsErrorId;
				nErrorId2 := fbSdoWrite.nSdoErrorId;
				nStateA_ResetError := 99;  //Error
			ELSE
				bGlobErrorReseted := TRUE;
				nStateA_ResetError := 0; //CheckGlobError
			END_IF
			fbSdoWrite(bExecute:= FALSE);
		END_IF
	//***************************End ResetGlobError***********************************
	
	//**********************Begin CheckAndResetAxisError******************************
	10:	//CheckAxisError
		nStateA_ResetError := 80; //Ready
		bGlobError := FALSE;
		FOR nAxisNr := 1 TO 7 BY 1 DO
			IF aFbZAxisRef[nAxisNr].stInput.nStatus.7 THEN //Achse vorhanden?
				aFbZAxisRef[nAxisNr].stStatus.bError := FALSE;
				//Restart Base erforderlich?
				IF 	aFbZAxisRef[nAxisNr].stInput.nError = 14 OR
					aFbZAxisRef[nAxisNr].stInput.nError = 15 OR
					aFbZAxisRef[nAxisNr].stInput.nError = 16 OR
					aFbZAxisRef[nAxisNr].stInput.nError = 24 OR
					aFbZAxisRef[nAxisNr].stInput.nError = 26 OR
					aFbZAxisRef[nAxisNr].stInput.nError = 254 THEN
					nStateA_ResetError := 20; //RestartMzBase
					RETURN;
				END_IF
				IF aFbZAxisRef[nAxisNr].stInput.nError > 0 OR aFbZAxisRef[nAxisNr].stInput.nStatus.3 THEN
					IF aFbZAxisRef[nAxisNr].stInput.nError = 22 OR aFbZAxisRef[nAxisNr].stInput.nError = 7THEN
						aFbZAxisRef[nAxisNr].stStatus.bIsHomed := FALSE;
					END_IF
					aFbZAxisRef[nAxisNr].stOutput.nMode := 0;
					aFbZAxisRef[nAxisNr].stOutput.nCtrl := 8;
					nStateA_ResetError := 11;
				END_IF
			END_IF
		END_FOR
	
	11:	//ControlByte zurücksetzen
		FOR nAxisNr := 1 TO 7 BY 1 DO
			IF aFbZAxisRef[nAxisNr].stInput.nStatus.7 THEN //Achse vorhanden?
				aFbZAxisRef[nAxisNr].stOutput.nCtrl := 0;	
			END_IF
		END_FOR
		tmrTimeout(IN:=FALSE);
		tmrTimeout(IN:=TRUE, PT:= T#500MS);
		nStateA_ResetError := 12;
		
	12: //Alle Achsen fehlerfrei?
		tmrTimeout();
		IF tmrTimeout.Q THEN
			tmrTimeout(IN:=FALSE);
			FOR nAxisNr := 1 TO 7 BY 1 DO
				IF aFbZAxisRef[nAxisNr].stInput.nStatus.7 THEN //Achse vorhanden?
					IF (aFbZAxisRef[nAxisNr].stInput.nError > 0 OR aFbZAxisRef[nAxisNr].stInput.nStatus.3) THEN
						//Fehler wurde nicht erfolgreich zurückgesetzt -> MzBase neu starten
						nStateA_ResetError := 20; //RestartMzBase
						RETURN;
					END_IF
				END_IF
			END_FOR
			nStateA_ResetError := 0; //CheckGlobError
			bGlobErrorReseted := FALSE;
		END_IF
	//***********************End CheckAndResetAxisError*******************************
	
	//***************************Begin RestartMzBase**********************************
	20: //Restart MzBase durch setzen von UpdateRequest
		//Ctrl und Mode der aller Achsen zurücksetzen
		FOR nAxisNr := 1 TO 7 BY 1 DO
			aFbZAxisRef[nAxisNr].stOutput.nCtrl := 0;
			aFbZAxisRef[nAxisNr].stOutput.nMode := 0;
			aFbZAxisRef[nAxisNr].stStatus.bIsHomed := FALSE;
		END_FOR
	
		IF bMzBaseRestarted THEN //Wurde MzBase bereits 1x neu gestarted, dann in Error gehen
			nErrorId := E_ErrorIdCmd.ERRORID_ErrorResetFailed;
			nErrorId2 := 0;
			nStateA_ResetError := 99;  //Error
		ELSE
			fbSdoWrite(sADSNetID:= stAdsAdress.sNetId, nPortNr:= stAdsAdress.nPort,
						nIndex:= cUpdateRequest.nIndex, nSubIndex:= cUpdateRequest.nSubIndex, 
						nDataLength:= cUpdateRequest.nLength, nData:= 1, bExecute:= TRUE);
						
			IF NOT fbSdoWrite.bBusy THEN
				IF fbSdoWrite.bError THEN
					nErrorId := fbSdoWrite.nAdsErrorId;
					nErrorId2 := fbSdoWrite.nSdoErrorId;
					nStateA_ResetError := 99;  //Error
				ELSE
					nStateA_ResetError := 21;
				END_IF
				fbSdoWrite(bExecute:= FALSE);
			END_IF
		END_IF
	
	21:	//Warten, bis NodeState von MzBase ungleich "0"
		IF nNodeState > 0 THEN
			tmrTimeout(IN:= FALSE);
			nStateA_ResetError := 22;
		END_IF
		
	22:	//Warten, bis MzBase sich wieder meldet und auf operational geht
		tmrTimeout(IN:= TRUE,PT:= T#6S);
		IF tmrTimeout.Q THEN
			nErrorId := E_ErrorIdCan.ERRORID_NodeNotFound;
			nStateA_ResetError := 99;  //Error
		END_IF
	
		IF nNodeState = 0 THEN
			nStateA_ResetError := 0; //CheckGlobError
			bMzBaseRestarted := TRUE;
			//Falls MzBase neugestartet wurde und es tritt nachher wieder ein Fehler auf
			//dann in ErrorState gehen
		END_IF
	//***************************End RestartMzBase***********************************
END_CASE

//**************************BeginError**********************************
IF nStateA_ResetError = 99 THEN
	fbErrorList.M_AddExt(nErrorId:= nErrorId, nErrorId2:= nErrorId2, 
	HardwareGrp:= E_HardwareGrp.AxisZ, 
	HardwareNr:= 0, 
	POU:= E_POU.POU_FB_MultiZRef, 
	POUAction:= E_POUACT.POUACT_A_Reset,
	POUState:= nPOUState);
	nErrorId2 := 0;
END_IF
//***************************EndError***********************************
END_ACTION

ACTION A_SetConfig:
stError.POUState := nStateA_SetConfig;
IF nStateA_SetConfig = 0 THEN	//nächste Achse ermitteln
	nStateA_SetConfig := 80;
	FOR nAxisNr := nAxisNr + 1 TO 7 BY 1 DO
		//Achse vorhanden?
		IF aFbZAxisRef[nAxisNr].stInput.nStatus.7 THEN
			IF aFbZAxisRef[nAxisNr].bIsSubAxis AND aFbZAxisRef[nAxisNr].bHasTool THEN
				stError.ErrorId := E_ErrorIdMultiZ.ERRORID_InvalidToolConfig;
				stError.ErrorId2 := 0;
				nStateA_SetConfig := 99;			
			ELSE
				stError.HardwareNr := nAxisNr;
				IF aFbZAxisRef[nAxisNr].bHasTool AND NOT(aFbZAxisRef[nAxisNr].eFixedToolType = E_MzToolType.TOOL_TYPE_None) THEN
					nStateA_SetConfig := 1; //weiter zu Vergleich ToolType
				ELSE
					nStateA_SetConfig := 0;
				END_IF				
			END_IF
			EXIT;
		ELSE
			IF aFbZAxisRef[nAxisNr].bHasTool THEN
				stError.ErrorId := E_ErrorIdMultiZ.ERRORID_NoZAxis;
				nStateA_SetConfig := 99;
				EXIT;
			END_IF
		END_IF			
	END_FOR
END_IF

IF nStateA_SetConfig = 1 THEN	//ToolType vergleichen
	//Bei allen Tools außer den generischen, muss einfach auf Gleichheit überprüft werden
	IF aFbZAxisRef[nAxisNr].eDetectedToolType = E_MzToolType.TOOL_TYPE_GenericPEXTool THEN
		IF aFbZAxisRef[nAxisNr].eFixedToolType = E_MzToolType.TOOL_TYPE_TipEjector OR 
			aFbZAxisRef[nAxisNr].eFixedToolType = E_MzToolType.TOOL_TYPE_PowderPip THEN
			nStateA_SetConfig := 2;
		ELSE
			stError.ErrorId := E_ErrorIdMultiZ.ERRORID_InvalidToolConfig;
			stError.ErrorId2 := 0;
			nStateA_SetConfig := 99;
		END_IF
	ELSIF aFbZAxisRef[nAxisNr].eDetectedToolType = aFbZAxisRef[nAxisNr].eFixedToolType THEN
		nStateA_SetConfig := 0;
	ELSIF aFbZAxisRef[nAxisNr].eDetectedToolType = E_MzToolType.TOOL_TYPE_PiezoSingle THEN
		IF aFbZAxisRef[nAxisNr].eFixedToolType = E_MzToolType.TOOL_TYPE_PiezoPip THEN
			nStateA_SetConfig := 0;
		ELSE
			stError.ErrorId := E_ErrorIdMultiZ.ERRORID_InvalidToolConfig;
			stError.ErrorId2 := 0;
			nStateA_SetConfig := 99;
		END_IF
	ELSIF aFbZAxisRef[nAxisNr].eDetectedToolType = E_MzToolType.TOOL_TYPE_PowderPipGen2 THEN
		nStateA_SetConfig := 0;
	ELSE
		stError.ErrorId := E_ErrorIdMultiZ.ERRORID_InvalidToolConfig;
		stError.ErrorId2 := 0;
		nStateA_SetConfig := 99;		
	END_IF
END_IF

IF nStateA_SetConfig = 2 THEN	//ToolType bei GenericTools überschreiben
	fbSdoWrite(sADSNetID:= stAdsAdress.sNetId, nPortNr:= stAdsAdress.nPort,
				nIndex:= cToolType.nIndex, nSubIndex := nAxisNr, nDataLength:= cToolType.nLength,
				nData := aFbZAxisRef[nAxisNr].eFixedToolType, bExecute:= TRUE);
	IF NOT fbSdoWrite.bBusy THEN
		IF fbSdoWrite.bError THEN
			stError.ErrorId := fbSdoWrite.nAdsErrorId;
			stError.ErrorId2 := fbSdoWrite.nSdoErrorId;
			nStateA_SetConfig := 99;  //Error
		ELSE
			nStateA_SetConfig := 0;
		END_IF
		fbSdoWrite(bExecute:= FALSE);
	END_IF
END_IF

IF nStateA_SetConfig = 99 THEN
	stError.Cmd := 0;
	stError.HardwareGrp := E_HardwareGrp.AxisZ;
	stError.POU := E_POU.POU_FB_MultiZRef;
	stError.POUAction := E_POUACT.POUACT_A_SetConfig;
	fbErrorList.M_Add(stError);
END_IF
END_ACTION

ACTION A_SetConfigLegacy:
//Wenn sich die lokale und remote ToolChecksum unterscheiden, dann MultiZ resetten
CASE nStateA_SetConfig OF
	0: //RemoteCrc auslesen
		fbSdoRead(sADSNetID:= stAdsAdress.sNetId, nPortNr:= stAdsAdress.nPort, 
					nIndex:= cConfigCRC.nIndex, nSubIndex:= cConfigCRC.nSubIndex,
					nDataLength:= cConfigCRC.nLength, bExecute:= TRUE);
		IF NOT fbSdoRead.bBusy THEN
			IF fbSdoRead.bError THEN
				nErrorId := fbSdoRead.nAdsErrorId;
				nErrorId2 := fbSdoRead.nSdoErrorId;
				nStateA_SetConfig := 99;
			ELSE
				nLocalCRC := M_GetToolChecksum();
				nRemoteCRC := DINT_TO_UINT(fbSdoRead.nData);
				IF nLocalCRC = 16#A96A THEN //braucht nicht konfiguriert werden da keine aktiven Tools vorhanden
					nStateA_SetConfig := 80;		
				ELSE
					IF nRemoteCRC = 0 THEN //wurde noch nicht konfiguriert
						nStateA_SetConfig := 4;	//konfigurieren ohne zu resetten
					ELSIF nLocalCRC = nRemoteCRC THEN //Konfiguration ist identisch
						nStateA_SetConfig := 80;
					ELSE
						nStateA_SetConfig := 1;	//Reset MultiZ, anschließend konfigurieren
					END_IF
				END_IF
			END_IF
			fbSdoRead(bExecute:= FALSE);
		END_IF
	
	1:	//MultiZ resetten
		P_bStopMonitor := TRUE;
		fbSdoWrite.nIndex := cUpdateRequest.nIndex;
		fbSdoWrite.nSubIndex := cUpdateRequest.nSubIndex;
		fbSdoWrite.nDataLength := cUpdateRequest.nLength;
		fbSdoWrite.nData := 1;
		nStateA_SetConfigNext := 2;
		nStateA_SetConfig := 50;
		
	2:	//Warten, bis sich MultiZ wieder meldet
		tmrTimeout(IN:= TRUE, PT:= T#6S);
		IF tmrTimeout.Q THEN
			tmrTimeout(IN:= FALSE);
			nStateA_SetConfig := 99;
		END_IF
		IF nNodeState = 0 THEN
			tmrTimeout(IN:= FALSE);
			nStateA_SetConfig := 3;
		END_IF
		
	3:	//Warten bis MultiZ bereit zum konfigurieren
		tmrTimeout(IN:= TRUE, PT:= T#1000MS);
		IF tmrTimeout.Q THEN
			tmrTimeout(IN:= FALSE);
			nStateA_SetConfig := 4;
		END_IF
END_CASE

IF nStateA_SetConfig = 4 THEN //nächste Achse ermitteln
	nAxisNr := nAxisNr + 1;
	IF nAxisNr = 8 THEN
		IF bSetConfigEnable THEN
			nStateA_SetConfig := 40;
			RETURN;
		ELSE
			bSetConfigEnable := TRUE;
			nAxisNr := 1;
		END_IF
	END_IF

	//Checken, ob Achse vorhanden
	IF aFbZAxisRef[nAxisNr].stInput.nStatus.7 THEN
		IF bSetConfigEnable THEN
			IF aFbZAxisRef[nAxisNr].eFixedToolType <> E_MzToolType.TOOL_TYPE_None THEN //ToolEnable setzen
				aFbZAxisRef[nAxisNr].stOutput.nToolEnable := 1;
				fbSdoWrite.nIndex := cToolEnable.nIndex;
				fbSdoWrite.nSubIndex := nAxisNr;
				fbSdoWrite.nDataLength := cToolEnable.nLength;
				fbSdoWrite.nData := 1;
				nStateA_SetConfig := 50; //SdoSend
				nStateA_SetConfigNext := 4;
			END_IF
		ELSE
			CASE aFbZAxisRef[nAxisNr].eFixedToolType OF
				E_MzToolType.TOOL_TYPE_Cartridge,E_MzToolType.TOOL_TYPE_PiezoPip,E_MzToolType.TOOL_TYPE_TipEjector,E_MzToolType.TOOL_TYPE_Stamp, E_MzToolType.TOOL_TYPE_PowderPip:
				IF aFbZAxisRef[nAxisNr].eFixedToolType = E_MzToolType.TOOL_TYPE_Stamp THEN
					aFbZAxisRef[nAxisNr + 1].bIsSubAxis := TRUE;
					aFbZAxisRef[nAxisNr + 2].bIsSubAxis := TRUE;
				END_IF
					nStateA_SetConfig := 5; //ToolType setzen
			ELSE
				RETURN;
			END_CASE
		END_IF
	ELSE
		RETURN;
	END_IF
END_IF

CASE nStateA_SetConfig OF
	5:	//ToolType setzen
		fbSdoWrite.nIndex := cToolType.nIndex;
		fbSdoWrite.nSubIndex := nAxisNr;
		fbSdoWrite.nDataLength := cToolType.nLength;
		fbSdoWrite.nData := aFbZAxisRef[nAxisNr].eFixedToolType;
		nStateA_SetConfigNext := 6;
		nStateA_SetConfig := 50; //SdoSend
		
	6:	//HeaterExist setzen
		fbSdoWrite.nIndex := cHeaterExist.nIndex;
		fbSdoWrite.nSubIndex := nAxisNr;
		fbSdoWrite.nDataLength := cHeaterExist.nLength;
		fbSdoWrite.nData := BOOL_TO_DINT(aFbHeaterRef[nAxisNr].P_bHeaterFixed);
		nStateA_SetConfigNext := 4; //nächste Achse
		nStateA_SetConfig := 50; //SdoSend
		
	40:	//Checken, ob MultiZ einen globalen Fehler bringt
		CASE nErrorGlobal OF
			8,14,18,255:
				nErrorId := F_MultiZError_TO_ErrorId(nErrorGlobal);
				nStateA_SetConfig := 99;  //Error wird im FB geworfen
		ELSE
			//FixConfig setzen
			bFixConfig := TRUE;
			fbSdoWrite.nIndex := cConfigFix.nIndex;
			fbSdoWrite.nSubIndex := cConfigFix.nSubIndex;
			fbSdoWrite.nDataLength := cConfigFix.nLength;
			fbSdoWrite.nData := 1;
			nStateA_SetConfigNext := 41;
			nStateA_SetConfig := 50;
		END_CASE
	
	41: //Die Achsen, bei denen das ToolEnable gesetzt ist, müssen innerhalb einerhalb des Timeouts
		//das Bit3 von ToolState bringen
		nStateA_SetConfig := 42;
		tmrTimeout(IN:= TRUE, PT:=T#1S);
		FOR nAxisNr := 1 TO 7 BY 1 DO
			IF aFbZAxisRef[nAxisNr].stOutput.nToolEnable = 1 THEN
				IF NOT aFbZAxisRef[nAxisNr].stInput.nToolState.3 THEN
					nStateA_SetConfig := 41;
					EXIT;
				END_IF
			END_IF
		END_FOR
		IF tmrTimeout.Q THEN
			nStateA_SetConfig := 42;
			tmrTimeout(IN:= FALSE);
		END_IF
			
	42:	//Checken, ob alle Achsen fehlerfrei
		nStateA_SetConfig := 43;
		FOR nAxisNr := 1 TO 7 BY 1 DO
			IF aFbZAxisRef[nAxisNr].stInput.nError > 0 THEN
				nErrorId := aFbZAxisRef[nAxisNr].stInput.nError;
				nStateA_SetConfig := 99;  //Error wird im FB geworfen
			END_IF
		END_FOR
		
	43:	
		bMzBaseRestarted := FALSE;
		P_bStopMonitor := FALSE;
		nStateA_SetConfig := 80;
END_CASE

//SDO senden
IF nStateA_SetConfig = 50 THEN
	fbSdoWrite(sADSNetID:= stAdsAdress.sNetId, nPortNr:= stAdsAdress.nPort, bExecute:= TRUE);
	IF NOT fbSdoWrite.bBusy THEN
		IF fbSdoWrite.bError THEN
			nErrorId := fbSdoWrite.nAdsErrorId;
			nErrorId2 := fbSdoWrite.nSdoErrorId;
			nStateA_SetConfig := 99;  //Error
		ELSE
			nStateA_SetConfig := nStateA_SetConfigNext;
		END_IF
		fbSdoWrite(bExecute:= FALSE);
	END_IF			
END_IF
END_ACTION

METHOD FB_init : BOOL
VAR_INPUT
	bInitRetains : BOOL; // if TRUE, the retain variables are initialized (warm start / cold start)
	bInCopyCode : BOOL;  // if TRUE, the instance afterwards gets moved into the copy code (online change)
END_VAR
stHardwareId.eGroup := E_HardwareGrp.MultiZBasis;
END_METHOD

METHOD M_DelConfig
VAR_INPUT
END_VAR
FOR nAxisNr := 1 TO 7 BY 1 DO
	aFbZAxisRef[nAxisNr].bHasTool := FALSE;
	aFbZAxisRef[nAxisNr].eFixedToolType := E_MzToolType.TOOL_TYPE_None;
	//aFbZAxisRef[nAxisNr].bIsSubAxis := FALSE;
	aFbHeaterRef[nAxisNr].P_bHeaterDetected := FALSE;
END_FOR
END_METHOD

METHOD M_GetHwInfo : ST_HardwareInfo
VAR_INPUT
END_VAR
M_GetHwInfo := SUPER^.M_GetHwInfo();
M_GetHwInfo.sSoftwVersion2 := USINT_TO_STRING(nTriggerVersion);
END_METHOD

METHOD M_GetPiezoRef : POINTER TO FB_PiezoRef
VAR_INPUT
	nChannel : USINT;
END_VAR
IF nChannel > 0 AND nChannel <= 7 THEN
	M_GetPiezoRef := ADR(aFbPiezoRef[nChannel]);
END_IF
END_METHOD

METHOD M_GetToolChecksum : UINT
VAR_INPUT
END_VAR
VAR
	i : USINT;
	nToolType : UINT;
	nHeater	: UINT;
	nResult : UINT;
	wPrevChecksum	: UINT := 16#FFFF;
END_VAR
//Diese Funktion wird nur bei Kopfbasisplatine ohne Toolerkennung benötigt
FOR i:= 1 TO 7 BY 1 DO
	nToolType := SHL(USINT_TO_UINT(aFbZAxisRef[i].eFixedToolType),8); 
	nHeater := BOOL_TO_UINT(aFbHeaterRef[i].P_bHeaterFixed);
	nResult := nToolType OR nHeater;
	wPrevChecksum := F_DATA_TO_CRC16_CCITT(ADR(nResult),SIZEOF(nResult),wPrevChecksum);
END_FOR
M_GetToolChecksum := wPrevChecksum;
END_METHOD

METHOD M_GetZSensorCalib : REAL
VAR_INPUT
	nZSensorId : DINT;
	nAxisNr : USINT;
END_VAR

VAR
	i : USINT;
END_VAR
FOR i := 1 TO 4 BY 1 DO
	IF stZSensorCalibration[i].nId = nZSensorId AND stZSensorCalibration[i].nAxis = nAxisNr THEN //Eintrag gefunden
		M_GetZSensorCalib := stZSensorCalibration[i].rValue;
		RETURN;
	END_IF
END_FOR
END_METHOD

METHOD M_Reset
VAR_INPUT
END_VAR
IF bError AND NOT bBusy THEN
	bBusy := TRUE;
	bResetError := TRUE;
	bMzBaseRestarted := FALSE;
END_IF
END_METHOD

METHOD M_SetConfig : ERRORID
VAR_INPUT
END_VAR
IF NOT (bBusy OR bSetConfig) THEN
	nAxisNr := 0;
	bSetConfigEnable := FALSE;
	bBusy := TRUE;
	bSetConfig := TRUE;
END_IF
END_METHOD

METHOD M_SetDigiOut : BOOL
VAR_INPUT
	nChannel : USINT;
	bValue : BOOL;
END_VAR
IF nChannel > 0 AND nChannel < 8 THEN
	aDigiOut[nChannel] := bValue;
	M_SetDigiOut := TRUE;
END_IF
END_METHOD

METHOD M_SetZSensorCalib
VAR_INPUT
	nZSensorId : DINT;
	nAxisNr : USINT;
	rValue : REAL;	
END_VAR

VAR
	i : USINT;
	nFree : USINT;
	bFound : BOOL;
END_VAR
//vorhandenen Eintrag suchen
FOR i := 1 TO 4 BY 1 DO
	IF stZSensorCalibration[i].nId = 0 THEN //kein Eintrag
		IF nFree = 0 THEN
			nFree := i; //erste freie Zeile
		END_IF
	ELSIF stZSensorCalibration[i].nId = nZSensorId AND stZSensorCalibration[i].nAxis = nAxisNr THEN //Eintrag gefunden
		stZSensorCalibration[i].rValue := rValue;
		fbSettings.M_WritePersData(); //Daten persitent schreiben
		bFound := TRUE;
		RETURN;
	END_IF
END_FOR

IF NOT bFound THEN //es wurde kein Eintrag gefunden
	IF nFree = 0 THEN //keine freie Zeile vorhanden, ersten Eintrag überschreiben und folgende nach hinten verschieben
		stZSensorCalibration[4] := stZSensorCalibration[3];
		stZSensorCalibration[3] := stZSensorCalibration[2];
		stZSensorCalibration[2] := stZSensorCalibration[1];
		stZSensorCalibration[1].nId := nZSensorId;
		stZSensorCalibration[1].nAxis := nAxisNr;
		stZSensorCalibration[1].rValue := rValue;
		fbSettings.M_WritePersData(); //Daten persitent schreiben
	ELSE
		stZSensorCalibration[nFree].nId := nZSensorId;
		stZSensorCalibration[nFree].nAxis := nAxisNr;
		stZSensorCalibration[nFree].rValue := rValue;
		fbSettings.M_WritePersData(); //Daten persitent schreiben
	END_IF
END_IF
END_METHOD

PROPERTY P_bLegacy : BOOL
GET
P_bLegacy := bLegacy;
END_GET
END_PROPERTY

PROPERTY P_bMzBaseRestarted : BOOL
GET
P_bMzBaseRestarted := bMzBaseRestarted;
END_GET
END_PROPERTY

PROPERTY P_nAdsPort : UINT
GET
P_nAdsPort := stAdsAdress.nPort;
END_GET
END_PROPERTY

PROPERTY P_nAxisNrZSensor : USINT
GET
P_nAxisNrZSensor := nAxisNrZSensor;
END_GET
SET
nAxisNrZSensor := P_nAxisNrZSensor;
END_SET
END_PROPERTY

PROPERTY P_nTriggerVersion : USINT
GET
P_nTriggerVersion := nTriggerVersion;
END_GET
END_PROPERTY

PROPERTY P_stError : ST_Error
GET
P_stError := stError;
END_GET
END_PROPERTY

END_FUNCTION_BLOCK

// ---- Hardware/MultiZ/FB_ZAxisRef.TcPOU
FUNCTION_BLOCK FB_ZAxisRef EXTENDS FB_HwModule
VAR_INPUT
	stInput 			: ST_ZAxisRef_In;
	stOutput 			: ST_ZAxisRef_Out;
	stStatus			: ST_ZAxisStatus;
	
	eDetectedToolType 	: E_MzToolType; //Sdo , wird nur bei Kopfbasisplatinen mir Toolerkennung benutzt und wird bei 
										//A_PrepareAxis in FB_MultiZRef ausgelesen
	eFixedToolType		: E_MzToolType; //Sdo, wird in den Objekten gesetzt und dann in A_SetConfig oder A_SetConfigLegacy
										//in FB_MultiZRef ausgelesen 
	
	bHasTool	: BOOL;
	sTmcVersion	: STRING(5);
	nTmcModulId	: UINT;
	nToolVersion: USINT;
	bIsSubAxis	: BOOL; //Ist eine Unterachse z.B. vom Stempel (wird vom Stempel gesteuert)
	bIngoreError: BOOL; //verhindert das Abfangen eines Fehlers in "A_Monitor"
	pCurrentFb	: POINTER TO PVOID;
END_VAR

VAR_OUTPUT
	pMultiZRef : POINTER TO FB_MultiZRef;
	nChannel : USINT;
END_VAR

VAR PERSISTENT
	rMaxSpeed 		: REAL;
	rRefPos 		: REAL;
	rMaxPos			: REAL;
	rMinPos			: REAL;
	rHomePos		: REAL;
	rAxisLength		: REAL;
	rSliderLength	: REAL;
	bInvertInitDir	: BOOL;
END_VAR

VAR
	nZSensorID  : DINT;
END_VAR

METHOD FB_init : BOOL
VAR_INPUT
	bInitRetains : BOOL; // if TRUE, the retain variables are initialized (warm start / cold start)
	bInCopyCode : BOOL;  // if TRUE, the instance afterwards gets moved into the copy code (online change)
	pMultiZRef : POINTER TO FB_MultiZRef;
END_VAR

VAR
	nFirstAdress : PVOID;
	nSelfAdress : PVOID;
END_VAR
THIS^.pMultiZRef := pMultiZRef;
nFirstAdress := ADR(pMultiZRef^.aFbZAxisRef);
nSelfAdress := THIS;
{IF hasvalue (RegisterSize, '32')}
nChannel := UDINT_TO_USINT((nSelfAdress - nFirstAdress)/SIZEOF(THIS^) + 1);
{ELSE}
nChannel := ULINT_TO_USINT((nSelfAdress - nFirstAdress)/SIZEOF(THIS^) + 1);
{END_IF}
stHardwareId.eGroup := E_HardwareGrp.AxisZ;
stHardwareId.nItem := nChannel;
END_METHOD

METHOD M_GetHwInfo : ST_HardwareInfo
VAR_INPUT
END_VAR
M_GetHwInfo := SUPER^.M_GetHwInfo();
M_GetHwInfo.sHardwVersion := UINT_TO_STRING(nTmcModulId);
M_GetHwInfo.sSoftwVersion := sTmcVersion;
M_GetHwInfo.sSoftwVersion2 := USINT_TO_STRING(nToolVersion);
END_METHOD

METHOD M_RenewHwId
VAR_INPUT
END_VAR

VAR
	stHwIdParent : ST_HardwareId;
END_VAR
stHwIdParent := pMultiZRef^.P_stHardwareId;
stHardwareId.nParentItem := stHwIdParent.nItem;
END_METHOD

PROPERTY P_bInvertInitDir : BOOL
GET
P_bInvertInitDir := bInvertInitDir;
END_GET
SET
bInvertInitDir := P_bInvertInitDir;
fbSettings.M_WritePersData();
END_SET
END_PROPERTY

PROPERTY P_nZSensorID : DINT
GET
P_nZSensorID := nZSensorID;
END_GET
SET
nZSensorID := P_nZSensorID;
END_SET
END_PROPERTY

PROPERTY P_rAbsTargetPos : REAL
SET
stOutput.nTrgtPos := REAL_TO_DINT(rAxisLength - rSliderLength - P_rAbsTargetPos);
END_SET
END_PROPERTY

PROPERTY P_rAxisLength : REAL
GET
P_rAxisLength := rAxisLength;
END_GET
SET
rAxisLength := P_rAxisLength;
fbSettings.M_WritePersData();
END_SET
END_PROPERTY

PROPERTY P_rCurrentPos : REAL
GET
P_rCurrentPos := MIN(rAxisLength - rSliderLength - DINT_TO_REAL(stInput.nCurrentPos),rMaxPos);
END_GET
END_PROPERTY

PROPERTY P_rHomePos : REAL
GET
P_rHomePos := rHomePos;
END_GET
SET
rHomePos := P_rHomePos;
fbSettings.M_WritePersData();
END_SET
END_PROPERTY

PROPERTY P_rMaxPos : REAL
GET
P_rMaxPos := rMaxPos;
END_GET
SET
rMaxPos := P_rMaxPos;
END_SET
END_PROPERTY

PROPERTY P_rMaxSpeed : REAL
GET
P_rMaxSpeed := rMaxSpeed;
END_GET
SET
rMaxSpeed := P_rMaxSpeed;
fbSettings.M_WritePersData();
END_SET
END_PROPERTY

PROPERTY P_rMinPos : REAL
GET
P_rMinPos := rMinPos;
END_GET
SET
rMinPos := P_rMinPos;
fbSettings.M_WritePersData();
END_SET
END_PROPERTY

PROPERTY P_rRefPos : REAL
GET
P_rRefPos := rRefPos;
END_GET
SET
rRefPos := P_rRefPos;
fbSettings.M_WritePersData();
END_SET
END_PROPERTY

PROPERTY P_rRelTargetPos : REAL
SET
stOutput.nTrgtPos := REAL_TO_DINT(- P_rRelTargetPos);
END_SET
END_PROPERTY

PROPERTY P_rSliderLength : REAL
GET
P_rSliderLength := rSliderLength;
END_GET
SET
rSliderLength := P_rSliderLength;
fbSettings.M_WritePersData();
END_SET
END_PROPERTY

PROPERTY P_rSpeed : REAL
GET
END_GET
SET
END_SET
END_PROPERTY

END_FUNCTION_BLOCK

// ---- Hardware/MultiZ/Piezo/FB_PiezoRef.TcPOU
FUNCTION_BLOCK FB_PiezoRef
VAR_INPUT
END_VAR
VAR
	nPeriod			: UINT;
	nPulse			: UINT;
	nDrops			: UINT;
	nVoltage		: UINT;
	nHoldVoltage	: UINT;
	nPrePeakTime	: UINT;
	nZSensorID  	: DINT;
	eDispenserMode 	: E_DispenserMode;
	bSynchronize	: BOOL;
END_VAR

VAR_OUTPUT
	pMultiZRef 	: POINTER TO FB_MultiZRef;
	nChannel 	: USINT;
	pToolCtrl	: POINTER TO BYTE;
	pToolState	: POINTER TO BYTE;
END_VAR

METHOD FB_init : BOOL
VAR_INPUT
	bInitRetains 	: BOOL; // if TRUE, the retain variables are initialized (warm start / cold start)
	bInCopyCode 	: BOOL;  // if TRUE, the instance afterwards gets moved into the copy code (online change)
	pMultiZRef 		: POINTER TO FB_MultiZRef;
END_VAR

VAR
	nFirstAdress : PVOID;
	nSelfAdress : PVOID;		
END_VAR
THIS^.pMultiZRef := pMultiZRef;
nFirstAdress := ADR(pMultiZRef^.aFbPiezoRef);
nSelfAdress := THIS;
{IF hasvalue (RegisterSize, '32')}
nChannel := UDINT_TO_USINT((nSelfAdress - nFirstAdress)/SIZEOF(THIS^) + 1);
{ELSE}
nChannel := ULINT_TO_USINT((nSelfAdress - nFirstAdress)/SIZEOF(THIS^) + 1);
{END_IF}
pToolCtrl := ADR(pMultiZRef^.aFbZAxisRef[nChannel].stOutput.nToolCtrl);
pToolState := ADR(pMultiZRef^.aFbZAxisRef[nChannel].stInput.nToolState);
END_METHOD

PROPERTY P_bSynchronize : BOOL
GET
P_bSynchronize := bSynchronize;
END_GET
SET
bSynchronize := P_bSynchronize;
END_SET
END_PROPERTY

PROPERTY P_eDispenserMode : E_DispenserMode
GET
P_eDispenserMode := eDispenserMode;
END_GET
SET
eDispenserMode := P_eDispenserMode;
END_SET
END_PROPERTY

PROPERTY P_nDrops : UINT
GET
P_nDrops := nDrops;
END_GET
SET
nDrops := P_nDrops;
END_SET
END_PROPERTY

PROPERTY P_nHoldVoltage : UINT
GET
P_nHoldVoltage := nHoldVoltage;
END_GET
SET
nHoldVoltage := P_nHoldVoltage;
END_SET
END_PROPERTY

PROPERTY P_nPeriod : UINT
GET
P_nPeriod := nPeriod;
END_GET
SET
nPeriod := P_nPeriod;
END_SET
END_PROPERTY

PROPERTY P_nPrePeakTime : UINT
GET
P_nPrePeakTime := nPrePeakTime;
END_GET
SET
nPrePeakTime := P_nPrePeakTime;
END_SET
END_PROPERTY

PROPERTY P_nPulse : UINT
GET
P_nPulse := nPulse;
END_GET
SET
nPulse := P_nPulse;
END_SET
END_PROPERTY

PROPERTY P_nVoltage : UINT
GET
P_nVoltage := nVoltage;
END_GET
SET
 nVoltage := P_nVoltage;
END_SET
END_PROPERTY

PROPERTY P_nZSensorID : DINT
GET
P_nZSensorID := nZSensorID;
END_GET
END_PROPERTY

END_FUNCTION_BLOCK

// ---- Hardware/MultiZ/Heater/FB_MZHeaterRef.TcPOU
FUNCTION_BLOCK FB_MZHeaterRef
VAR_INPUT
END_VAR
VAR_OUTPUT
	pMultiZRef 		: POINTER TO FB_MultiZRef;
	nChannel 		: USINT;
	nTemp1Actual 	AT %I* : UINT;
	nTemp2Actual 	AT %I* : UINT;
	nTemp3Actual 	AT %I* : UINT;	
	bHeaterIsOn		AT %I* : BOOL;
END_VAR
VAR
	bHeaterExistDetected	: BOOL;
	bHeaterExistFixed		: BOOL;
	nTemp1Setpoint	: UINT;
END_VAR

METHOD FB_init : BOOL
VAR_INPUT
	bInitRetains : BOOL; // if TRUE, the retain variables are initialized (warm start / cold start)
	bInCopyCode : BOOL;  // if TRUE, the instance afterwards gets moved into the copy code (online change)
	pMultiZRef 		: POINTER TO FB_MultiZRef;
END_VAR

VAR
	nFirstAdress : PVOID;
	nSelfAdress : PVOID;
END_VAR
THIS^.pMultiZRef := pMultiZRef;
nFirstAdress := ADR(pMultiZRef^.aFbHeaterRef);
nSelfAdress := THIS;
{IF hasvalue (RegisterSize, '32')}
nChannel := UDINT_TO_USINT((nSelfAdress - nFirstAdress)/SIZEOF(THIS^) + 1);
{ELSE}
nChannel := ULINT_TO_USINT((nSelfAdress - nFirstAdress)/SIZEOF(THIS^) + 1);
{END_IF}
END_METHOD

PROPERTY P_bHeaterDetected : BOOL
GET
P_bHeaterDetected := bHeaterExistDetected;
END_GET
SET
bHeaterExistDetected := P_bHeaterDetected;
END_SET
END_PROPERTY

PROPERTY P_bHeaterFixed : BOOL
GET
P_bHeaterFixed := bHeaterExistFixed;
END_GET
SET
bHeaterExistFixed := P_bHeaterFixed;
END_SET
END_PROPERTY

PROPERTY P_nTemp1Setpoint : UINT
GET
P_nTemp1Setpoint := nTemp1Setpoint;
END_GET
SET
nTemp1Setpoint := P_nTemp1Setpoint;
END_SET
END_PROPERTY

END_FUNCTION_BLOCK

// ---- Hardware/MultiZ/Extruder/FB_PistonExtruderRef.TcPOU
FUNCTION_BLOCK FB_PistonExtruderRef EXTENDS FB_ExtruderRef
VAR_INPUT
END_VAR
VAR
	nCurrentPlungerPos 	AT %I* : DINT;
	bLimitSwitch		AT %I* : BOOL;
	
	nUnlockOffsetOrgin	: DINT; //µm
	nUnlockOffsetCalc	: DINT; //µm
END_VAR

VAR_OUTPUT
	pMultiZRef 	: POINTER TO FB_MultiZRef;
	nChannel 	: USINT;
	pToolCtrl	: POINTER TO BYTE;
	pToolState	: POINTER TO BYTE;
END_VAR

METHOD FB_init : BOOL
VAR_INPUT
	bInitRetains : BOOL; // if TRUE, the retain variables are initialized (warm start / cold start)
	bInCopyCode : BOOL;  // if TRUE, the instance afterwards gets moved into the copy code (online change)
	pMultiZRef 		: POINTER TO FB_MultiZRef;
END_VAR

VAR
	nFirstAdress : PVOID;
	nSelfAdress : PVOID;
END_VAR
THIS^.pMultiZRef := pMultiZRef;
nFirstAdress := ADR(pMultiZRef^.aFbExtruderRef);
nSelfAdress := THIS;
{IF  hasvalue (RegisterSize, '32')}
nChannel := UDINT_TO_USINT((nSelfAdress - nFirstAdress)/SIZEOF(THIS^) + 1);
{ELSE}
nChannel := ULINT_TO_USINT((nSelfAdress - nFirstAdress)/SIZEOF(THIS^) + 1);
{END_IF}
pToolCtrl := ADR(pMultiZRef^.aFbZAxisRef[nChannel].stOutput.nToolCtrl);
pToolState := ADR(pMultiZRef^.aFbZAxisRef[nChannel].stInput.nToolState);
END_METHOD

PROPERTY P_bError : BOOL
GET
P_bError := (pMultiZRef^.aFbZAxisRef[nChannel].stInput.nError > 0);
END_GET
END_PROPERTY

PROPERTY P_bIsActive : BOOL
GET
P_bIsActive := pToolState^.0;
END_GET
END_PROPERTY

PROPERTY P_bIsLocked : BOOL
GET
P_bIsLocked := pToolState^.4;
END_GET
END_PROPERTY

PROPERTY P_nCurrentPos : DINT
GET
P_nCurrentPos := REAL_TO_DINT(DINT_TO_REAL(nCurrentPlungerPos) / rFactorDistance);
END_GET
END_PROPERTY

PROPERTY P_nUnlockOffsetCalc : DINT
GET
P_nUnlockOffsetCalc := nUnlockOffsetCalc;
END_GET
END_PROPERTY

PROPERTY P_nUnlockOffsetOrgin : DINT
GET
P_nUnlockOffsetOrgin := nUnlockOffsetOrgin;
END_GET
SET
nUnlockOffsetOrgin := P_nUnlockOffsetOrgin;
nUnlockOffsetCalc := REAL_TO_DINT(rFactorDistance * DINT_TO_REAL(nUnlockOffsetOrgin));
END_SET
END_PROPERTY

END_FUNCTION_BLOCK

// ---- Hardware/MultiZ/Extruder/FB_ExtruderRef.TcPOU
FUNCTION_BLOCK FB_ExtruderRef
VAR_INPUT
END_VAR
VAR
	rFactorDistance		: REAL;
	rFactorFeed			: REAL;
	nFeedOrgin			: DINT;	//µm/s
	nCompFeedOrgin		: DINT;	//µm/s
	nRelaxFeedOrgin		: DINT;	//µm/s
	nDistanceOrgin		: DINT;	//µm
	nCompDistanceOrgin	: DINT;	//µm
	nRelaxDistanceOrgin	: DINT;	//µm
	
	//Umgerechnete Werte
	nFeedCalc			: DINT; // 1/100tel RPM
	nCompFeedCalc		: DINT; // 1/100tel RPM
	nRelaxFeedCalc		: DINT; // 1/100tel RPM
	nDistanceCalc		: DINT;	// µm
	nCompDistanceCalc	: DINT;	// µm
	nRelaxDistanceCalc	: DINT;	// µm	
END_VAR
VAR_OUTPUT
END_VAR

//Basisklasse

PROPERTY P_bError : BOOL
GET
END_GET
END_PROPERTY

PROPERTY P_bIsActive : BOOL
GET
END_GET
END_PROPERTY

PROPERTY P_bIsLocked : BOOL
GET
END_GET
END_PROPERTY

PROPERTY P_nCompDistanceCalc : DINT
GET
P_nCompDistanceCalc := nCompDistanceCalc;
END_GET
END_PROPERTY

PROPERTY P_nCompDistanceOrgin : DINT
GET
P_nCompDistanceOrgin := nCompDistanceOrgin;
END_GET
SET
nCompDistanceOrgin := P_nCompDistanceOrgin;
nCompDistanceCalc := REAL_TO_DINT(rFactorDistance * DINT_TO_REAL(nCompDistanceOrgin));
END_SET
END_PROPERTY

PROPERTY P_nCompFeedCalc : DINT
GET
P_nCompFeedCalc := nCompFeedCalc;
END_GET
END_PROPERTY

PROPERTY P_nCompFeedOrgin : DINT
GET
P_nCompFeedOrgin := nCompFeedOrgin;
END_GET
SET
nCompFeedOrgin := P_nCompFeedOrgin;
nCompFeedCalc := REAL_TO_DINT(rFactorFeed * DINT_TO_REAL(nCompFeedOrgin));
END_SET
END_PROPERTY

PROPERTY P_nCurrentPos : DINT
GET
END_GET
END_PROPERTY

PROPERTY P_nDistanceCalc : DINT
GET
P_nDistanceCalc := nDistanceCalc;
END_GET
END_PROPERTY

PROPERTY P_nDistanceOrgin : DINT
GET
P_nDistanceOrgin := nDistanceOrgin;
END_GET
SET
nDistanceOrgin := P_nDistanceOrgin;
nDistanceCalc := REAL_TO_DINT(rFactorDistance * DINT_TO_REAL(nDistanceOrgin));
END_SET
END_PROPERTY

PROPERTY P_nFeedCalc : DINT
GET
P_nFeedCalc := nFeedCalc;
END_GET
END_PROPERTY

PROPERTY P_nFeedOrgin : DINT
GET
P_nFeedOrgin := nFeedOrgin;
END_GET
SET
nFeedOrgin := P_nFeedOrgin;
nFeedCalc := REAL_TO_DINT(rFactorFeed * DINT_TO_REAL(nFeedOrgin));
END_SET
END_PROPERTY

PROPERTY P_nRelaxDistanceCalc : DINT
GET
P_nRelaxDistanceCalc := nRelaxDistanceCalc;
END_GET
END_PROPERTY

PROPERTY P_nRelaxDistanceOrgin : DINT
GET
P_nRelaxDistanceOrgin := nRelaxDistanceOrgin;
END_GET
SET
nRelaxDistanceOrgin := P_nRelaxDistanceOrgin;
nRelaxDistanceCalc := REAL_TO_DINT(rFactorDistance * DINT_TO_REAL(nRelaxDistanceOrgin));
END_SET
END_PROPERTY

PROPERTY P_nRelaxFeedCalc : DINT
GET
P_nRelaxFeedCalc := nRelaxFeedCalc;
END_GET
END_PROPERTY

PROPERTY P_nRelaxFeedOrgin : DINT
GET
P_nRelaxFeedOrgin := nRelaxFeedOrgin;
END_GET
SET
nRelaxFeedOrgin := P_nRelaxFeedOrgin;
nRelaxFeedCalc := REAL_TO_DINT(rFactorFeed * DINT_TO_REAL(nRelaxFeedOrgin));
END_SET
END_PROPERTY

PROPERTY P_rFactorDistance : REAL
GET
P_rFactorDistance := rFactorDistance;
END_GET
SET
rFactorDistance := P_rFactorDistance;
END_SET
END_PROPERTY

PROPERTY P_rFactorFeed : REAL
GET
P_rFactorFeed := rFactorFeed;
END_GET
SET
rFactorFeed := P_rFactorFeed;
END_SET
END_PROPERTY

END_FUNCTION_BLOCK

// ---- Hardware/MultiZ/Gripper/FB_GripperRef.TcPOU
FUNCTION_BLOCK FB_GripperRef
VAR_INPUT
END_VAR
VAR_OUTPUT
END_VAR
VAR
	nChannel 		: USINT;
	pToolCtrl		: POINTER TO BYTE;
	pToolState		: POINTER TO BYTE;
	bVialDetector	AT %I* : BOOL;
END_VAR

METHOD FB_init : BOOL
VAR_INPUT
	bInitRetains 	: BOOL; // if TRUE, the retain variables are initialized (warm start / cold start)
	bInCopyCode 	: BOOL;  // if TRUE, the instance afterwards gets moved into the copy code (online change)
	pMultiZRef 		: POINTER TO FB_MultiZRef;
END_VAR

VAR
	nFirstAdress : PVOID;
	nSelfAdress : PVOID;		
END_VAR
nFirstAdress := ADR(pMultiZRef^.aFbGripperRef);
nSelfAdress := THIS;
{IF hasvalue (RegisterSize, '32')}
nChannel := UDINT_TO_USINT((nSelfAdress - nFirstAdress)/SIZEOF(THIS^) + 1);
{ELSE}
nChannel := ULINT_TO_USINT((nSelfAdress - nFirstAdress)/SIZEOF(THIS^) + 1);
{END_IF}
pToolCtrl := ADR(pMultiZRef^.aFbZAxisRef[nChannel].stOutput.nToolCtrl);
pToolState := ADR(pMultiZRef^.aFbZAxisRef[nChannel].stInput.nToolState);
END_METHOD

METHOD M_Actuate
VAR_INPUT
	eCtrl : E_OpClCtrl;
END_VAR
pToolCtrl^ := eCtrl;
END_METHOD

PROPERTY P_bVialDetector : BOOL
GET
P_bVialDetector := NOT bVialDetector;
END_GET
END_PROPERTY

PROPERTY P_eGripperState : E_GripperState
GET
IF pToolState^ = 24 THEN
	P_eGripperState := E_GripperState.Open;
ELSIF pToolState^ = 9 THEN
	P_eGripperState := E_GripperState.HalfClosed;
ELSIF pToolState^ = 11 THEN
	P_eGripperState := E_GripperState.FullyClosed;
ELSE
	P_eGripperState := E_GripperState.Undefined;
END_IF
END_GET
END_PROPERTY

END_FUNCTION_BLOCK

// ---- Hardware/MultiZ/GPIO/FB_GPInputRef.TcPOU
FUNCTION_BLOCK FB_GPInputRef
VAR_INPUT
	bInit	: BOOL;
	eMode : E_GPInputMode;
END_VAR
VAR_OUTPUT
	pMultiZRef 		: POINTER TO FB_MultiZRef;
	nChannel 		: USINT;
	nValue			AT %I* : UINT;
	bBusy			: BOOL;
	bError			: BOOL;
	nErrorId		: ERRORID;
END_VAR
VAR
	nState : USINT;
	fbSdoWrite : FB_SDO_WRITE;
END_VAR

IF bInit THEN
	IF nState = 0 THEN
		fbSdoWrite(sADSNetID:= pMultiZRef^.P_sAdsNetId, nPortNr:= pMultiZRef^.P_nAdsPort, 
					nIndex:= cGPInputMode.nIndex , nSubIndex:= nChannel, nDataLength:= cGPInputMode.nLength, nData:= eMode, bExecute:= TRUE);
		IF NOT fbSdoWrite.bBusy THEN
			IF fbSdoWrite.bError THEN
				bError := TRUE;
				nErrorId := fbSdoWrite.nAdsErrorId;
				nState := 99;
			ELSE
				nState := 80;
			END_IF
 			fbSdoWrite(bExecute := FALSE); 
		END_IF
	END_IF
ELSE
	bError := FALSE;
	nErrorId := 0;
	nState := 0;
END_IF

METHOD FB_init : BOOL
VAR_INPUT
	bInitRetains : BOOL; // if TRUE, the retain variables are initialized (warm start / cold start)
	bInCopyCode : BOOL;  // if TRUE, the instance afterwards gets moved into the copy code (online change)
	pMultiZRef 	: POINTER TO FB_MultiZRef;
END_VAR

VAR
	nFirstAdress : PVOID;
	nSelfAdress : PVOID;
END_VAR
THIS^.pMultiZRef := pMultiZRef;
nFirstAdress := ADR(pMultiZRef^.aFbGPInputRef);
nSelfAdress := THIS;
{IF hasvalue (RegisterSize, '32')}
nChannel := UDINT_TO_USINT((nSelfAdress - nFirstAdress)/SIZEOF(THIS^) + 1);
{ELSE}
nChannel := ULINT_TO_USINT((nSelfAdress - nFirstAdress)/SIZEOF(THIS^) + 1);
{END_IF}
END_METHOD

END_FUNCTION_BLOCK

// ---- Hardware/MultiZ/F_MultiZError_TO_ErrorId.TcPOU
FUNCTION F_MultiZError_TO_ErrorId : ERRORID
VAR_INPUT
	nErrorCode	: USINT;
END_VAR
VAR
END_VAR

F_MultiZError_TO_ErrorId := nErrorCode + 41727;

END_FUNCTION

// ---- Hardware/F_CompVersion.TcPOU
FUNCTION F_CompVersion : SINT
VAR_INPUT
	sVersion1 : STRING;
	sVersion2 : STRING;
END_VAR
VAR
	nChar	: BYTE;
	aVersion1 : ARRAY[0..2] OF UINT;
	aVersion2 : ARRAY[0..2] OF UINT;
	i : INT;
	j : USINT;
	sTemp	: STRING;
END_VAR

//Version1 in Array einlesen
FOR i:= 0 TO LEN(sVersion1) BY 1 DO
	nChar := sVersion1[i];
	IF nChar >= 48 AND nChar <= 57 THEN //numerisch
		sTemp := CONCAT(sTemp,F_ToCHR(nChar));
	ELSIF nChar = 46 OR nChar = 32 OR nChar = 0 THEN //Punkt Leerzeichen oder ENDE
		aVersion1[j] := STRING_TO_UINT(sTemp);
		sTemp := '';
		j := j + 1;
		IF j = 3 THEN
			EXIT;
		END_IF
	END_IF
END_FOR
//Version2 in Array einlesen
j := 0;
sTemp := '';
FOR i:= 0 TO LEN(sVersion2) BY 1 DO
	nChar := sVersion2[i];
	IF nChar >= 48 AND nChar <= 57 THEN //numerisch
		sTemp := CONCAT(sTemp,F_ToCHR(nChar));
	ELSIF nChar = 46 OR nChar = 32 OR nChar = 0 THEN //Punkt Leerzeichen oder ENDE
		aVersion2[j] := STRING_TO_UINT(sTemp);
		sTemp := '';
		j := j + 1;
		IF j = 3 THEN
			EXIT;
		END_IF
	END_IF
END_FOR

FOR i:= 2 TO 0 BY -1 DO
	IF aVersion1[i] < aVersion2[i] THEN
		F_CompVersion := -1;
	ELSIF aVersion1[i] > aVersion2[i] THEN
		F_CompVersion := 1;
	END_IF
END_FOR

END_FUNCTION

// ---- Objects/Targets/FB_TargetBase.TcPOU
FUNCTION_BLOCK FB_TargetBase EXTENDS FB_Object
VAR_INPUT
END_VAR
VAR_OUTPUT
END_VAR
VAR
	//Targetproperties
	pParentTarget		: POINTER TO FB_TargetBase;
	stRelPos 			: ST_3DPoint;
	stDimension			: ST_3DDimension;
	rFreeHeight			: REAL;
	rZOffset			: REAL;
	nCurrentPropIndex	: UINT;
	nSpecPropIndex		: UINT;			//erster Index für Specialproperties (ab direkter Erbe von FB_MzTool) (benötigt in M_SetSingleProps + M_GetSingleProp)
END_VAR

METHOD M_AddChild : ERRORID
VAR_INPUT
	pObject	: POINTER TO FB_Object;
	nSlotNr	: UINT;
	nIndex 	: INT;	
END_VAR
//In den abgeleiteten Tool-FBs wird überprüft, ob das entsprechende Objekt als Child tauglich ist
IF pObject > 0 THEN
	IF nSlotNr = 0 THEN
		//Object darf selber noch an keinem Parent hängen
		IF pObject^.P_pParentObject = 0 THEN
			pObject^.P_pObjCollectNode := pObjCollectNode^.nodes.M_AddNewNode(pObject,nIndex);
			pObject^.M_UpdateParent();
		ELSE
			M_AddChild := E_ErrorIdObjMgmt.ERRORID_ObjectAlreadyOnAnotherParent;
		END_IF
	ELSE
		M_AddChild := E_ErrorIdObjMgmt.ERRORID_InvalidSlotNumber;			
	END_IF	
ELSE
	M_AddChild := E_ErrorIdObjMgmt.ERRORID_InvalidParentObject;
END_IF
END_METHOD

METHOD M_ApplyPos : ERRORID
VAR_INPUT
	eTargetRef 		: E_TargetRef;
	nPointSlotNr	: UINT;
	stPos 			: ST_3DPoint;
	bXPos			: BOOL;
	bYPos			: BOOL;
	bZPos			: BOOL;	
END_VAR

VAR
	stParentPos	: ST_3DPoint;
END_VAR
//Neue relative Position berechen
//ZOffset (gemessener Wert wird auf "0" gesetzt) 
rZOffset := 0;
IF pParentTarget > 0 THEN
	stParentPos := pParentTarget^.P_stAbsPosLB;
	IF pParentSlot > 0 THEN
		stParentPos := F_Add3DPoints(stParentPos,pParentSlot^.P_stRelPos);
	END_IF
END_IF

CASE eTargetRef OF
	E_TargetRef.TARGETREF_LeftBottom:
		IF bXPos THEN
			stRelPos.X := stPos.X - stParentPos.X;	
		END_IF
		IF bYPos THEN
			stRelPos.Y := stPos.Y - stParentPos.Y;	
		END_IF
		IF bZPos THEN
			stRelPos.Z := stPos.Z - stParentPos.Z - stDimension.Height;
			P_pWorkplate^.P_bCalcCollisHeight := TRUE;		
		END_IF
	E_TargetRef.TARGETREF_LeftTop:
		IF bXPos THEN
			stRelPos.X := stPos.X - stParentPos.X;	
		END_IF
		IF bYPos THEN
			stRelPos.Y := stPos.Y - stParentPos.Y - stDimension.Depth;	
		END_IF
		IF bZPos THEN
			stRelPos.Z := stPos.Z - stParentPos.Z - stDimension.Height;	
			P_pWorkplate^.P_bCalcCollisHeight := TRUE;
		END_IF
	E_TargetRef.TARGETREF_RightTop:
		IF bXPos THEN
			stRelPos.X := stPos.X - stParentPos.X - stDimension.Width;	
		END_IF
		IF bYPos THEN
			stRelPos.Y := stPos.Y - stParentPos.Y - stDimension.Depth;	
		END_IF
		IF bZPos THEN
			stRelPos.Z := stPos.Z - stParentPos.Z - stDimension.Height;	
		END_IF
	E_TargetRef.TARGETREF_RightBottom:
		IF bXPos THEN
			stRelPos.X := stPos.X - stParentPos.X - stDimension.Width;	
		END_IF
		IF bYPos THEN
			stRelPos.Y := stPos.Y - stParentPos.Y;	
		END_IF
		IF bZPos THEN
			stRelPos.Z := stPos.Z - stParentPos.Z - stDimension.Height;
			P_pWorkplate^.P_bCalcCollisHeight := TRUE;
		END_IF
	E_TargetRef.TARGETREF_Center:
		IF bXPos THEN
			stRelPos.X := stPos.X - stParentPos.X - stDimension.Width / 2.0;	
		END_IF
		IF bYPos THEN
			stRelPos.Y := stPos.Y - stParentPos.Y - stDimension.Depth / 2.0;	
		END_IF
		IF bZPos THEN
			stRelPos.Z := stPos.Z - stParentPos.Z - stDimension.Height;
			P_pWorkplate^.P_bCalcCollisHeight := TRUE;
		END_IF
END_CASE
END_METHOD

METHOD M_CheckAction : ERRORID
VAR_INPUT
	refActionData : REFERENCE TO ST_ActionData;
	pCorrelObject	: POINTER TO FB_Object;
END_VAR
IF refActionData.eAction = E_Action.ACTION_TeachTarget THEN
	IF NOT eObjectType = E_ObjectType.OBJECTTYPE_Point AND DINT_TO_UINT(refActionData.aParams[1]) = E_TargetRef.TARGETREF_Center THEN
		M_CheckAction := E_ErrorIdCmd.ERRORID_InvalidTargetPointRef; 
	END_IF
END_IF
END_METHOD

METHOD M_CheckProps : ERRORID
VAR_INPUT
END_VAR
END_METHOD

METHOD M_ClearAllProps
VAR_INPUT
	bIgnoreParent : BOOL; //Es wird das gesamte OD gelöscht. -> Zeiger auf Parent nicht mehr gültig!
END_VAR
IF NOT bIgnoreParent THEN
	IF pParentSlot > 0 THEN
		pParentSlot^.P_pChild := 0;
	END_IF
END_IF

nObjectID := 0;
pParentTarget := 0;
pParentSlot := 0;
pObjCollectNode := 0;
END_METHOD

METHOD M_GetAbsPos : ST_3DPoint
VAR_INPUT
	pChildPos	: POINTER TO ST_3DPoint;
	eTargetRef 	: E_TargetRef;
	nParam1		: UINT;
 	nParam2		: UINT;
	nParam3		: USINT;
	nZLevel		: USINT;
END_VAR
VAR_OUTPUT
	nErrorId 	: ERRORID;
	lrAngle		: LREAL;
END_VAR
VAR
	stLocPos : ST_3DPoint;
	pSlot : POINTER TO FB_Slot;
END_VAR
stLocPos := stRelPos;
stLocPos.Z := stLocPos.Z + stDimension.Height + rZOffset;
CASE eTargetRef OF
	E_TargetRef.TARGETREF_LeftBottom:
		;
	E_TargetRef.TARGETREF_LeftTop:
		stLocPos.Y := stLocPos.Y + stDimension.Depth;
	E_TargetRef.TARGETREF_RightBottom:
		stLocPos.X := stLocPos.X + stDimension.Width;
	E_TargetRef.TARGETREF_RightTop:
		stLocPos.X := stLocPos.X + stDimension.Width;
		stLocPos.Y := stLocPos.Y + stDimension.Depth;
	E_TargetRef.TARGETREF_Center:
		stLocPos.X := stLocPos.X + stDimension.Width / 2.0;
		stLocPos.Y := stLocPos.Y + stDimension.Depth / 2.0;
ELSE
	nErrorId := E_ErrorIdCmd.ERRORID_InvalidTargetPointRef;
END_CASE

IF nErrorId > 0 THEN
	RETURN;
END_IF

IF pChildPos > 0 THEN
	stLocPos.X := stLocPos.X + pChildPos^.X;
	stLocPos.Y := stLocPos.Y + pChildPos^.Y;
	stLocPos.Z := stLocPos.Z + pChildPos^.Z;
END_IF

IF pParentTarget > 0 THEN
	IF pParentSlot > 0 THEN
 		stLocPos := pParentTarget^.M_GetAbsPos(pChildPos := ADR(stLocPos), eTargetRef:= E_TargetRef.TARGETREF_Slot,
													nParam1:= pParentSlot^.P_nNr,
													nParam2:= 0, nParam3:= 0,nZLevel:= 0, lrAngle=> lrAngle,
													nErrorId=> nErrorId);
	ELSE
 		stLocPos := pParentTarget^.M_GetAbsPos(pChildPos := ADR(stLocPos), eTargetRef:= E_TargetRef.TARGETREF_LeftBottom,
													nParam1:= 0,
													nParam2:= 0, nParam3:= 0,nZLevel:= 0, lrAngle=> lrAngle,
													nErrorId=> nErrorId);
	END_IF
END_IF

IF nErrorId > 0 THEN
	RETURN;
END_IF

M_GetAbsPos := stLocPos;
END_METHOD

METHOD M_GetAllProps : ERRORID
VAR_INPUT
	refCmdData : REFERENCE TO ST_CmdData;
END_VAR
refCmdData.aHeader[0] := nObjectID;
refCmdData.aHeader[1] := eObjectType;


//ParentTarget
IF pParentTarget > 0 THEN
	refCmdData.n32Data[0] := pParentTarget^.P_nObjectID;
END_IF

//ParentSlot
IF pParentSlot > 0 THEN
	refCmdData.n32Data[1] := pParentSlot^.P_nNr;
END_IF

//Relative Koordinaten lesen
refCmdData.n32Data[2] := REAL_TO_DINT(stRelPos.X);
refCmdData.n32Data[3] := REAL_TO_DINT(stRelPos.Y);
refCmdData.n32Data[4] := REAL_TO_DINT(stRelPos.Z);
//Dimensionen lesen
refCmdData.n32Data[5] := REAL_TO_DINT(stDimension.Width);
refCmdData.n32Data[6] := REAL_TO_DINT(stDimension.Depth);
refCmdData.n32Data[7] := REAL_TO_DINT(stDimension.Height);
refCmdData.n32Data[8] := REAL_TO_DINT(rFreeHeight);

nCurrentPropIndex := 8;

IF eObjectType = E_ObjectType.OBJECTTYPE_Point THEN
	refCmdData.n32Data[9] := REAL_TO_DINT(rZOffset);
	nCurrentPropIndex := 9;
END_IF
END_METHOD

METHOD M_GetFirstParentOfType : POINTER TO FB_TargetBase
VAR_INPUT
	eObjectType : E_ObjectType;
END_VAR
IF pParentTarget > 0 THEN
	IF pParentTarget^.P_eObjectType = eObjectType THEN
		M_GetFirstParentOfType := pParentTarget;
	ELSE
		M_GetFirstParentOfType := pParentTarget^.M_GetFirstParentOfType(eObjectType);
	END_IF
END_IF
END_METHOD

METHOD M_GetHighestTarget : POINTER TO FB_TargetBase
VAR_INPUT
	fbRectArea : FB_Rectangle;
	rHight : REAL;
END_VAR

VAR
	iter				: FB_ObjCollectIterator;
	pTarget 			: POINTER TO FB_TargetBase;
	fbRectTarget		: FB_Rectangle;
	bResult				: BOOL;
END_VAR
//Selber für sich checken, ob im Bereich
fbRectTarget := P_fbAbsRect;
IF F_RectInnerRect(fbRectTarget,fbRectArea) THEN
	bResult := TRUE; 
ELSIF F_RectInnerRect(fbRectArea,fbRectTarget) THEN
	bResult := TRUE;	
ELSIF F_LinesIntersect(fbRectTarget.P_LineBottom,fbRectArea.P_LineLeft) THEN
	bResult := TRUE;	
ELSIF F_LinesIntersect(fbRectTarget.P_LineBottom,fbRectArea.P_LineRight) THEN
	bResult := TRUE;	
ELSIF F_LinesIntersect(fbRectTarget.P_LineTop,fbRectArea.P_LineLeft) THEN
	bResult := TRUE;	
ELSIF F_LinesIntersect(fbRectTarget.P_LineTop,fbRectArea.P_LineRight) THEN
	bResult := TRUE;
ELSIF F_LinesIntersect(fbRectTarget.P_LineLeft,fbRectArea.P_LineBottom) THEN
	bResult := TRUE;
ELSIF F_LinesIntersect(fbRectTarget.P_LineLeft,fbRectArea.P_LineTop) THEN
	bResult := TRUE;
ELSIF F_LinesIntersect(fbRectTarget.P_LineRight,fbRectArea.P_LineBottom) THEN
	bResult := TRUE;
ELSIF F_LinesIntersect(fbRectTarget.P_LineRight,fbRectArea.P_LineTop) THEN
	bResult := TRUE;
ELSE
	bResult := FALSE;
END_IF

IF bResult THEN
	IF P_rAbsFreeHeight >= rHight THEN
		rHight := P_rAbsFreeHeight;
	END_IF
END_IF

//Childs durchlaufen

pObjCollectNode^.nodes.M_GetIterator(iter);
WHILE iter.pNode > 0 DO
	IF iter.pNode^.P_pObject > 0 AND_THEN iter.pNode^.P_pObject^.M_bIsGroup(E_ObjectGroup.OBJECTGROUP_Target) THEN
		pTarget := iter.pNode^.P_pObject;
		pTarget := pTarget^.M_GetHighestTarget(fbRectArea,rHight);
		IF pTarget > 0 THEN
			IF pTarget^.P_eObjectType <> E_ObjectType.OBJECTTYPE_Point THEN
				IF pTarget^.P_rAbsFreeHeight > rHight THEN
					M_GetHighestTarget := pTarget;
					rHight := pTarget^.P_rAbsFreeHeight;
				END_IF
			END_IF			
		END_IF
	END_IF
	iter.M_Increment();
END_WHILE

IF P_rAbsFreeHeight >= rHight AND bResult THEN
	M_GetHighestTarget := THIS;
END_IF
END_METHOD

METHOD M_GetPropCheckSum : UINT
VAR_INPUT
END_VAR

VAR
	stData 		: ST_CmdData;
END_VAR
M_GetAllProps(stData);
wChecksum := F_DATA_TO_CRC16_CCITT(ADR(stData.n32Data[0]),nNoOfProps * 4,16#FFFF);
M_GetPropCheckSum := wChecksum;
END_METHOD

METHOD M_IsPointInArea : BOOL
VAR_INPUT
	stPoint	: ST_3DPoint;
END_VAR

VAR
	stPointLB : ST_3DPoint;	//links unten
	stPointRT : ST_3DPoint;	//rechts oben
END_VAR


VAR_OUTPUT
	rAbsZ	: REAL;
END_VAR
stPointLB := P_stAbsPosLB;
stPointRT := P_stAbsPosRT;

IF stPoint.X >= stPointLB.X AND stPoint.X <= stPointRT.X AND stPoint.Y >= stPointLB.Y AND stPoint.Y <= stPointRT.Y THEN
	M_IsPointInArea := TRUE;
	rAbsZ := stPointLB.Z;
END_IF
END_METHOD

METHOD M_SetAllProps : ERRORID
VAR_INPUT
	refCmdData : REFERENCE TO  ST_CmdData;
END_VAR
nNoOfProps := 9;

//Relative Koordinaten setzen
stRelPos.X := DINT_TO_REAL(refCmdData.n32Data[2]);
stRelPos.Y := DINT_TO_REAL(refCmdData.n32Data[3]);
stRelPos.Z := DINT_TO_REAL(refCmdData.n32Data[4]);

//Dimensionen setzen
stDimension.Width := DINT_TO_REAL(refCmdData.n32Data[5]);
stDimension.Depth := DINT_TO_REAL(refCmdData.n32Data[6]);
stDimension.Height := DINT_TO_REAL(refCmdData.n32Data[7]);
rFreeHeight := DINT_TO_REAL(refCmdData.n32Data[8]);
nCurrentPropIndex := 8;

//Wenn ein Punkt, dann ZOffset
IF eObjectType = E_ObjectType.OBJECTTYPE_Point THEN
	nNoOfProps := 10;
	rZOffset := DINT_TO_REAL(refCmdData.n32Data[9]);
	nCurrentPropIndex := 9;
END_IF

P_pWorkplate^.P_bCalcCollisHeight := TRUE;
END_METHOD

METHOD M_SetSingleProp : ERRORID
VAR_INPUT
	refCmdData : REFERENCE TO  ST_CmdData;
END_VAR
//Basisproperties schreiben
CASE refCmdData.aHeader[1] OF	//Property-Nr
	2:	//XPosRel
		stRelPos.X := DINT_TO_REAL(refCmdData.n32Data[0]);
	3:	//YPosRel
		stRelPos.Y := DINT_TO_REAL(refCmdData.n32Data[0]);
	4:	//ZPosRel
		stRelPos.Z := DINT_TO_REAL(refCmdData.n32Data[0]);
		P_pWorkplate^.P_bCalcCollisHeight := TRUE;
	5:	//Width
		stDimension.Width := DINT_TO_REAL(refCmdData.n32Data[0]);
	6:	//Depth
		stDimension.Depth := DINT_TO_REAL(refCmdData.n32Data[0]);
	7:	//Height
		stDimension.Height := DINT_TO_REAL(refCmdData.n32Data[0]);
		P_pWorkplate^.P_bCalcCollisHeight := TRUE;
	8:	//FreeHeight
		rFreeHeight := DINT_TO_REAL(refCmdData.n32Data[0]);
		P_pWorkplate^.P_bCalcCollisHeight := TRUE;
	9:	
		//Wenn ein Punkt, dann ZOffset
		IF eObjectType = E_ObjectType.OBJECTTYPE_Point THEN
			rZOffset := DINT_TO_REAL(refCmdData.n32Data[0]);
			P_pWorkplate^.P_bCalcCollisHeight := TRUE;
		ELSE
			M_SetSingleProp := E_ErrorIdCmd.ERRORID_InvalidProperty;	
		END_IF
	ELSE
		//Ungültige Property-Nr
		M_SetSingleProp := E_ErrorIdCmd.ERRORID_InvalidProperty;
		RETURN;
END_CASE
END_METHOD

METHOD M_UpdateParent
VAR_INPUT
END_VAR

VAR
	pObject : POINTER TO FB_Object;
END_VAR
IF pObjCollectNode > 0 AND_THEN pObjCollectNode^.pOwnerColl > 0 THEN
	pObject := pObjCollectNode^.P_pOwnerColl^.pOwnerNode^.P_pObject;	
END_IF
 
IF pObject > 0 THEN
	pParentTarget := pObject;
	pParentSlot := pObject^.M_GetSlotFromChild(THIS);
ELSE
	pParentTarget := 0;
	pParentSlot := 0;
END_IF
END_METHOD

PROPERTY P_fbAbsRect : FB_Rectangle
GET
VAR
	stPoint	: ST_3DPoint;
END_VAR
stPoint := P_stAbsPosLB;
P_fbAbsRect.X1 := stPoint.X;
P_fbAbsRect.Y1 := stPoint.Y;
stPoint := P_stAbsPosRT;
P_fbAbsRect.X2 := stPoint.X;
P_fbAbsRect.Y2 := stPoint.Y;
END_GET
END_PROPERTY

PROPERTY P_lrAbsAngle : LREAL
GET
IF pParentTarget > 0 THEN
 P_lrAbsAngle := pParentTarget^.P_lrAbsAngle;
END_IF
END_GET
END_PROPERTY

PROPERTY P_nGCodeTargetNr : UINT
GET
(*IF pObjCollectNode > 0 AND eObjectGroup = OBJECTGROUP_Target THEN
	P_nGCodeTargetNr := P_nGCodeTargetNr +1;
	ELSE
		P_nGCodeTargetNr :=0;
	END_IF*)
END_GET
END_PROPERTY

PROPERTY P_pWorkplate : POINTER TO FB_Workplate
GET
IF eObjectType = E_ObjectType.OBJECTTYPE_Workplate THEN
	P_pWorkplate := THIS;
ELSE
	P_pWorkplate := pParentTarget^.P_pWorkplate;
END_IF
END_GET
END_PROPERTY

PROPERTY P_rAbsFreeHeight : REAL
GET
VAR
	stPoint : ST_3DPoint;
END_VAR
stPoint := P_stAbsPosCenter;
IF rFreeHeight > stDimension.Height THEN
	P_rAbsFreeHeight := stPoint.Z - stDimension.Height + rFreeHeight;
ELSE
	P_rAbsFreeHeight := stPoint.Z;
END_IF
END_GET
END_PROPERTY

PROPERTY P_rFreeHeight : REAL
GET
P_rFreeHeight := rFreeHeight;
END_GET
END_PROPERTY

PROPERTY P_rHeight : REAL
GET
P_rHeight := stDimension.Height;
END_GET
END_PROPERTY

PROPERTY P_rZOffset : REAL
GET
P_rZOffset := rZOffset;
END_GET
SET
rZOffset := P_rZOffset;
P_pWorkplate^.P_bCalcCollisHeight := TRUE;
END_SET
END_PROPERTY

PROPERTY P_stAbsPosCenter : ST_3DPoint	//Absolute Mitten-Position(XY) zum Workplate-Nullpunkt
GET
VAR
	stPosTmp	: ST_3DPoint;
END_VAR
stPosTmp.X := stDimension.Width / 2;
stPosTmp.Y := stDimension.Depth / 2;
stPosTmp.Z := stPosTmp.Z + stDimension.Height + P_rZOffset;
stPosTmp := F_Add3DPoints(stPosTmp,stRelPos);

IF pParentTarget > 0 THEN
	IF pParentSlot > 0 THEN
		P_stAbsPosCenter := F_Add3DPoints(pParentSlot^.P_stAbsPos, stPosTmp);
	ELSE
		P_stAbsPosCenter := F_Add3DPoints(pParentTarget^.P_stAbsPosLB, stPosTmp);	
	END_IF
ELSE
	P_stAbsPosCenter := stPosTmp;
END_IF
END_GET
END_PROPERTY

PROPERTY P_stAbsPosLB : ST_3DPoint
GET
VAR
	stPosTmp : ST_3DPoint;
END_VAR
IF pParentTarget > 0 THEN
	stPosTmp := stRelPos;
	stPosTmp.Z := stPosTmp.Z + stDimension.Height + P_rZOffset;
	IF pParentSlot > 0 THEN
		P_stAbsPosLB := F_Add3DPoints(pParentSlot^.P_stAbsPos,stPosTmp);
	ELSE
		P_stAbsPosLB := F_Add3DPoints(pParentTarget^.P_stAbsPosLB,stPosTmp);	
	END_IF
ELSE
	P_stAbsPosLB := stRelPos;
END_IF
END_GET
END_PROPERTY

PROPERTY P_stAbsPosLT : ST_3DPoint
GET
VAR
	stPosTmp : ST_3DPoint;
END_VAR
stPosTmp := stRelPos;
stPosTmp.Y := stPosTmp.Y + stDimension.Depth;
IF pParentTarget > 0 THEN
	stPosTmp.Z := stPosTmp.Z + stDimension.Height + P_rZOffset;
	IF pParentSlot > 0 THEN
		P_stAbsPosLT := F_Add3DPoints(pParentSlot^.P_stAbsPos,stPosTmp);
	ELSE
		P_stAbsPosLT := F_Add3DPoints(pParentTarget^.P_stAbsPosLB,stPosTmp);	
	END_IF
ELSE
	P_stAbsPosLT := stPosTmp;
END_IF
END_GET
END_PROPERTY

PROPERTY P_stAbsPosRB : ST_3DPoint	//Absolute Position zum Workplate-Nullpunkt (links unten)
GET
VAR
	stPosTmp : ST_3DPoint;
END_VAR
stPosTmp := stRelPos;
stPosTmp.X := stPosTmp.X + stDimension.Width;
IF pParentTarget > 0 THEN
	stPosTmp.Z := stPosTmp.Z + stDimension.Height + P_rZOffset;
	IF pParentSlot > 0 THEN
		P_stAbsPosRB := F_Add3DPoints(pParentSlot^.P_stAbsPos,stPosTmp);
	ELSE
		P_stAbsPosRB := F_Add3DPoints(pParentTarget^.P_stAbsPosLB,stPosTmp);	
	END_IF
ELSE
	P_stAbsPosRB := stPosTmp;
END_IF
END_GET
END_PROPERTY

PROPERTY P_stAbsPosRT : ST_3DPoint	//Absolute Position zum Workplate-Nullpunkt (links unten)
GET
VAR
	stPosTmp : ST_3DPoint;
END_VAR
stPosTmp := stRelPos;
stPosTmp.Y := stPosTmp.Y + stDimension.Depth;
stPosTmp.X := stPosTmp.X + stDimension.Width;
//IF nParentTargetIdx > 0 THEN
IF pParentTarget > 0 THEN
	stPosTmp.Z := stPosTmp.Z + stDimension.Height + P_rZOffset;
	IF pParentSlot > 0 THEN
		P_stAbsPosRT := F_Add3DPoints(pParentSlot^.P_stAbsPos,stPosTmp);
	ELSE
		P_stAbsPosRT := F_Add3DPoints(pParentTarget^.P_stAbsPosLB,stPosTmp);	
	END_IF
	
ELSE
	P_stAbsPosRT := stPosTmp;
END_IF
END_GET
END_PROPERTY

PROPERTY P_stAbsRect : ST_Rectangle
GET
VAR
	stPoint	: ST_3DPoint;
END_VAR
stPoint := P_stAbsPosLB;
P_stAbsRect.X1 := stPoint.X;
P_stAbsRect.Y1 := stPoint.Y;
stPoint := P_stAbsPosRT;
P_stAbsRect.X2 := stPoint.X;
P_stAbsRect.Y2 := stPoint.Y;
END_GET
END_PROPERTY

PROPERTY P_stDimension : ST_3DDimension
GET
P_stDimension := stDimension;
END_GET
SET
stDimension := P_stDimension;
P_pWorkplate^.P_bCalcCollisHeight := TRUE;
END_SET
END_PROPERTY

PROPERTY P_stRelPos : ST_3DPoint
GET
P_stRelPos := stRelPos;
END_GET
SET
stRelPos := P_stRelPos;
END_SET
END_PROPERTY

PROPERTY P_stRelPosLB : ST_3DPoint
GET
P_stRelPosLB := stRelPos;
P_stRelPosLB.Z := stRelPos.Z + stDimension.Height + rZOffset;
IF pParentTarget > 0 AND_THEN pParentSlot > 0 THEN
	P_stRelPosLB := F_Add3DPoints(P_stRelPosLB,pParentSlot^.P_stRelPos);
END_IF
END_GET
END_PROPERTY

END_FUNCTION_BLOCK

// ---- Objects/FB_Object.TcPOU
FUNCTION_BLOCK FB_Object
VAR_INPUT
END_VAR
VAR_OUTPUT
END_VAR
VAR
	nObjectID			: UINT;
	eObjectType 		: E_ObjectType;
	eObjectGroup		: E_ObjectGroup;//Zugehörigkeit zu Objektgruppe [Flags]
	pObjCollectNode		: POINTER TO FB_ObjCollectionNode;
	pParentSlot			: POINTER TO FB_Slot;
	nNoOfProps			: UINT;
	wChecksum			: WORD;
END_VAR

//Basisklasse für alle Objekte

METHOD M_AddChild : ERRORID
VAR_INPUT
	pObject	: POINTER TO FB_Object;
	nSlotNr	: UINT;
	nIndex : INT;
END_VAR
END_METHOD

METHOD M_bIsGroup : BOOL
VAR_INPUT
	eGroup	: E_ObjectGroup;
END_VAR
M_bIsGroup := (eObjectGroup AND eGroup) = eGroup;
END_METHOD

METHOD M_CheckProps : ERRORID
END_METHOD

METHOD M_ClearAllProps

VAR_INPUT
	bIgnoreParent : BOOL; //Es wird das gesamte OD gelöscht. -> Zeiger auf Parent nicht mehr gültig!
END_VAR
END_METHOD

METHOD M_GetAllProps : ERRORID
VAR_INPUT
	refCmdData	: REFERENCE TO ST_CmdData;
END_VAR
END_METHOD

METHOD M_GetDevice : I_Device
VAR_INPUT
END_VAR
END_METHOD

METHOD M_GetPropCheckSum : UINT
VAR_INPUT
END_VAR

VAR
	i			: UINT;
	stData 		: ST_CmdData;
END_VAR
M_GetAllProps(stData);
wChecksum := F_DATA_TO_CRC16_CCITT(ADR(stData.n32Data[0]),nNoOfProps * 4,16#FFFF);
M_GetPropCheckSum := wChecksum;
END_METHOD

METHOD M_GetSlot : POINTER TO FB_Slot
VAR_INPUT
	nSlotNr : UINT;
END_VAR
END_METHOD

METHOD M_GetSlotFromChild : POINTER TO FB_Slot
VAR_INPUT
	pObject : POINTER TO FB_Object;
END_VAR
END_METHOD

METHOD M_RemoveChild : ERRORID
VAR_INPUT
	pObject	: POINTER TO FB_Object;
END_VAR

VAR
	iter : FB_ObjCollectIterator;
END_VAR
//Das Objekt in der Collection suchen (flach)
pObjCollectNode^.nodes.M_GetIterator(iter);
WHILE iter.pNode > 0 DO
	IF iter.pNode^.P_pObject = pObject THEN
		//Falls Object an einem Slot, von diesem entfernen
		IF pObject^.P_pParentSlot > 0 THEN
			pObject^.P_pParentSlot^.P_pChild := 0;
		END_IF
		pObjCollectNode^.nodes.M_RemoveNode(iter.pNode);
		pObject^.M_UpdateParent();
		EXIT;
	END_IF
	iter.M_Increment();
END_WHILE

IF iter.pNode = 0 THEN
	M_RemoveChild := E_ErrorIdObjMgmt.ERRORID_ObjectNotInCollection;
END_IF
END_METHOD

METHOD M_SetAllProps : ERRORID
VAR_INPUT
	refCmdData	: REFERENCE TO ST_CmdData;
END_VAR
END_METHOD

METHOD M_SetSingleProp : ERRORID
VAR_INPUT
	refCmdData	: REFERENCE TO ST_CmdData;
END_VAR
END_METHOD

METHOD M_UpdateParent
END_METHOD

PROPERTY P_bHasChilds : BOOL
GET
P_bHasChilds := pObjCollectNode > 0 and_then pObjCollectNode^.nodes.nCount > 0;
END_GET
END_PROPERTY

PROPERTY P_eObjectGroup : E_ObjectGroup
GET
P_eObjectGroup := eObjectGroup;
END_GET
END_PROPERTY

PROPERTY P_eObjectType : E_ObjectType
GET
P_eObjectType := eObjectType;
END_GET
END_PROPERTY

PROPERTY P_nNoOfProps : UINT
GET
P_nNoOfProps := nNoOfProps;
END_GET
END_PROPERTY

PROPERTY P_nNotifyId : UINT
GET
END_GET
SET
END_SET
END_PROPERTY

PROPERTY P_nObjectID : UINT
GET
P_nObjectID := nObjectID;
END_GET
SET
nObjectID := P_nObjectID;
END_SET
END_PROPERTY

PROPERTY P_nParentSlotNr : UINT
GET
IF pParentSlot > 0 THEN
	P_nParentSlotNr := pParentSlot^.P_nNr;
END_IF
END_GET
END_PROPERTY

PROPERTY P_pObjCollectNode : POINTER TO FB_ObjCollectionNode
GET
P_pObjCollectNode := pObjCollectNode;
END_GET
SET
pObjCollectNode := P_pObjCollectNode;
END_SET
END_PROPERTY

PROPERTY P_pParentObject : POINTER TO FB_Object
GET
IF pObjCollectNode > 0 AND_THEN pObjCollectNode^.pOwnerColl > 0 AND_THEN pObjCollectNode^.pOwnerColl^.pOwnerNode > 0 THEN
	P_pParentObject := pObjCollectNode^.pOwnerColl^.pOwnerNode^.P_pObject;
END_IF
END_GET
END_PROPERTY

PROPERTY P_pParentSlot : POINTER TO FB_Slot
GET
P_pParentSlot := pParentSlot;
END_GET
END_PROPERTY

END_FUNCTION_BLOCK

// ---- Configuration/FB_ObjCollectionNode.TcPOU
{attribute 'enable_dynamic_creation'}
FUNCTION_BLOCK FB_ObjCollectionNode
VAR_INPUT
	pPrev : POINTER TO FB_ObjCollectionNode;
	pNext : POINTER TO FB_ObjCollectionNode;
END_VAR
VAR_OUTPUT
	nodes : FB_ObjCollection(THIS);
	pOwnerColl : POINTER TO FB_ObjCollection;
END_VAR
VAR
	pObject : POINTER TO FB_Object;
END_VAR

//Ist ein einzelnes Item einer Collection
//hat einen Vorgänger, Nachfolger, Parent(Collection), Nodes(Collection)

PROPERTY P_pOwnerColl : POINTER TO FB_ObjCollection
SET
pOwnerColl := P_pOwnerColl;
END_SET
GET
P_pOwnerColl := pOwnerColl;
END_GET
END_PROPERTY

PROPERTY P_pObject : POINTER TO FB_Object
GET
P_pObject := pObject;
END_GET
SET
pObject := P_pObject;
END_SET
END_PROPERTY

METHOD FB_init : BOOL
VAR_INPUT
	bInitRetains : BOOL; // if TRUE, the retain variables are initialized (warm start / cold start)
	bInCopyCode : BOOL;  // if TRUE, the instance afterwards gets moved into the copy code (online change)
	pOwnerColl : POINTER TO FB_ObjCollection;
END_VAR
THIS^.pOwnerColl := pOwnerColl;
END_METHOD

METHOD M_GetLevel : UINT
VAR_INPUT
	nStartLevel : UINT;
END_VAR
IF pOwnerColl^.pOwnerNode > 0 THEN
	nStartLevel := nStartLevel + 1;
	M_GetLevel := pOwnerColl^.pOwnerNode^.M_GetLevel(nStartLevel);
ELSE
	M_GetLevel := nStartLevel;
END_IF
END_METHOD

END_FUNCTION_BLOCK

// ---- Configuration/FB_ObjCollection.TcPOU
FUNCTION_BLOCK FB_ObjCollection
VAR_INPUT
END_VAR
VAR_OUTPUT
	nCount : UINT;
	pOwnerNode : POINTER TO FB_ObjCollectionNode;	//kann auch 0 sein wenn es die BasisCollection ist
END_VAR
VAR
	pHead : POINTER TO FB_ObjCollectionNode;
	pTail : POINTER TO FB_ObjCollectionNode;
END_VAR

//Soll es möglich sein, einen Node zu löschen, der nicht leer ist?
//Da sollte aber beachtet werden, dass es wenn es während einer Iteration gemacht wird, der Iterator eventuell nicht
//mehr gültig ist!
//für die richtige Anwendung soll es ja dann so sein, dass es ein flache Liste mit Devices gibt, die permanet ausgeführt
//werden. Es muss zwischen ObjectDirectory und dieser flachen Liste eine Verbindung geben, so dass wenn ein oder mehrere Nodes
//gelöscht werden, die Liste auch mit angepasst wird.

METHOD FB_init : BOOL
VAR_INPUT
	bInitRetains : BOOL; // if TRUE, the retain variables are initialized (warm start / cold start)
	bInCopyCode : BOOL;  // if TRUE, the instance afterwards gets moved into the copy code (online change)
	pOwnerNode : POINTER TO FB_ObjCollectionNode;
END_VAR
THIS^.pOwnerNode := pOwnerNode;
END_METHOD

METHOD M_AddExistNode
VAR_INPUT
	pNode : POINTER TO FB_ObjCollectionNode;
END_VAR

VAR
	
END_VAR
IF pHead = 0 THEN
	pHead := pTail := pNode;
ELSE
	pNode^.pPrev := pTail; 
	pTail^.pNext := pNode;
	pTail := pNode;	
END_IF
pNode^.P_pOwnerColl := THIS;
nCount := nCount + 1;
END_METHOD

METHOD M_AddNewNode : POINTER TO FB_ObjCollectionNode
VAR_INPUT
	pObject : POINTER TO FB_Object;
	nIndex : INT;
END_VAR

VAR
	pNew : POINTER TO FB_ObjCollectionNode;
	iter : FB_ObjCollectIterator;
	i : INT;
END_VAR
pNew := __NEW(FB_ObjCollectionNode(pOwnerColl:= THIS));
pNew^.P_pObject := pObject;
IF pHead = 0 THEN
	pHead := pTail := pNew;
ELSE
	//In Abhängigkeit vom Index an entsprechender Stelle einfügen oder ans Ende stellen
	IF nIndex < 0 OR INT_TO_UINT(nIndex) >= nCount THEN //am Ende anfügen
		pNew^.pPrev := pTail;
		pTail^.pNext := pNew;
		pTail := pNew;	
	ELSIF nIndex = 0 THEN //am Anfang einfügen
		pNew^.pNext := pHead;
		pHead^.pPrev := pNew;
		pHead := pNew;
	ELSE //vor das Element stellen, dass diesen Index jetzt hat
		//wenn es das Element nicht gibt, dann nichts machen
		//zuerst Element mit entsprechendem Index suchen
		M_GetIterator(iter);
		iter.M_Increment();
		WHILE iter.pNode > 0 DO
			i := i + 1; //beim ersten Durchlauf ist i = 1;
			//und man befindet sich hier bereits beim zweiten Node
			IF i = nIndex THEN
				//vor dem Node einfügen
				pNew^.pPrev := iter.pNode^.pPrev;
				pNew^.pPrev^.pNext := pNew;
				pNew^.pNext := iter.pNode;
				iter.pNode^.pPrev := pNew; 
				EXIT;
			END_IF
			iter.M_Increment();
		END_WHILE
	END_IF
END_IF
nCount := nCount + 1;
M_AddNewNode := pNew;
END_METHOD

METHOD M_Clear
VAR_INPUT
END_VAR

VAR
	iter : FB_ObjCollectIterator;
	pNode : POINTER TO FB_ObjCollectionNode;		
END_VAR
//alle Nodes und deren Childs löschen!
//das geht nur rekursiv
M_GetIterator(Iterator:= iter);
WHILE iter.pNode > 0 DO
	iter.pNode^.nodes.M_Clear();
	pNode := iter.pNode;
	iter.M_Increment();
	__DELETE(pNode);
	nCount := nCount - 1;
END_WHILE
pHead := 0;
pTail := 0;
END_METHOD

METHOD M_ClearNode
VAR_INPUT
	pNode : POINTER TO FB_ObjCollectionNode;
END_VAR

VAR
	iter : FB_ObjCollectIterator;
END_VAR
IF pNode > 0 AND_THEN pNode^.nodes.nCount = 0 THEN
	M_GetIterator(iter);
	WHILE iter.pNode > 0 DO
		IF pNode = iter.pNode THEN
			IF pNode = pHead THEN
				pHead := pHead^.pNext;
				IF pHead > 0 THEN
					pHead^.pPrev := 0;
				ELSE
					pTail := 0;
				END_IF
			ELSIF pNode = pTail THEN
				pTail := pTail^.pPrev;
				pTail^.pNext := 0;	
			ELSE
				pNode^.pPrev^.pNext := pNode^.pNext;
				pNode^.pNext^.pPrev := pNode^.pPrev;
			END_IF
			nCount := nCount - 1;
			__DELETE(pNode);
			EXIT;
		END_IF
		iter.M_Increment();
	END_WHILE
END_IF
END_METHOD

METHOD M_FindNode : POINTER TO FB_ObjCollectionNode
VAR_INPUT
	pNode : POINTER TO FB_ObjCollectionNode;
END_VAR

VAR
	iter : FB_ObjCollectIteratorDeep;
END_VAR
//Knoten in diesem und den unteren Bäumen suchen
IF pNode > 0 THEN
	M_GetIterator(Iterator:= iter);
	WHILE iter.pNode > 0 DO
		IF iter.pNode = pNode THEN
			M_FindNode := iter.pNode;
			RETURN; 	
		END_IF
		iter.M_Increment();
	END_WHILE
END_IF
END_METHOD

METHOD M_GetIterator
VAR_IN_OUT
	Iterator : FB_ObjCollectIterator;
END_VAR
Iterator(pInitNode := pHead);
END_METHOD

METHOD M_RemoveNode
VAR_INPUT
	pNode : POINTER TO FB_ObjCollectionNode;
END_VAR

